// TwinCAT 3 PLC project DeviceLib
// Title: IBF_Device
// Company: Industrial Brains B.V.
// ProjectVersion: 0.0.0.0
// ProgramVersion: 3.1.4022.4
// CompilerDefines: InclSerialCom := 'true'
// libraries:
//   IBF_Utilities, * (Industrial Brains B.V.)
//   Tc2_Math, * (Beckhoff Automation GmbH)
//   Tc2_MC2, * (Beckhoff Automation GmbH)
//   Tc2_MC2_Drive, * (Beckhoff Automation GmbH)
//   Tc2_Standard, * (Beckhoff Automation GmbH)
// project tree:
//   Actuators/Cylinder/DataTypes/ E_CylinderCmd.TcTLEO, E_ValveResetState.TcTLEO
//   Actuators/Cylinder/DataTypes/ManualControls/ UDT_ManualValveControl.TcDUT
//   Actuators/Cylinder/Functions/ Fb_DevCylWithFbk.TcPOU, FB_DevValve.TcPOU
//   Axis/DataTypes/ E_AxisCmd.TcTLEO, UDT_AxisData.TcDUT, UDT_AxVal.TcDUT, UDT_ManualAxisCtrl.TcDUT
//   Axis/FunctionBlocks/Analog/ FB_DevAnalogAxis.TcPOU, ST_ManualAnalogAxisCtrl.TcDUT (not stored)
//   Axis/FunctionBlocks/ServoHybrid/ FB_DevBasicACAxis.TcPOU, FB_DevHybridAc.TcPOU
//   Axis/FunctionBlocks/Servo/ Fb_DevAxis.TcPOU
//   Axis/FunctionBlocks/TwoVelocityControl/DataTypes/ st_ManualDigitalMotorControl.TcDUT (not stored)
//   Axis/FunctionBlocks/TwoVelocityControl/ FB_DevTwoVelocityAxis.TcPOU
//   Axis/Interface/ iTwoDirectionalMotor.TcIO (not stored), iTwoDirectionalMotorWithFast.TcIO (not stored)
//   BaseFunctions/ FB_DevBase.TcPOU, UDT_DevManualCtrl.TcDUT
//   Buttons/Functions/ FB_DevHMIButton.TcPOU, FB_DevPushbuttonLight.TcPOU, FB_DevPushButton.TcPOU
//   CounterCards/FunctionBlocks/KL1512/ FB_DevKL1512.TcPOU
//   CounterCards/FunctionBlocks/KL5151/ FB_DevKL5151.TcPOU
//   CounterCards/Interfaces/ iCounter.TcIO
//   CounterCards/ st_ManualCounterControl.TcDUT
//   DevTypes/ E_Devices.TcTLEO
//   Encoders/FunctionBlocks/ FB_EncoderBase.TcPOU, FB_EncoderInput.TcPOU
//   GroupHandlers/ GVL_DevManual.TcGVL
//   GroupHandlers/ManualControlHandler/ FB_ManualController.TcPOU, UDT_DeviceID.TcDUT
//   HardwareDiagnostics/ FB_ELModuleDiag.TcPOU
//   Heaters/ FB_DevDoublePWM.TcPOU, FB_DevPWMGenerator.TcPOU
//   Lights/Functions/ Fb_DevLight.TcPOU
//   Outputs/AnalogOutputs/ FB_DevAnalogOutput.TcPOU, FB_DevAnalogOutputScaled.TcPOU
//   Outputs/DigitalOutputs/ FB_DevDigitalOutput.TcPOU
//   Sensors/AnalogInput/FunctionBlocks/ FB_DevAnalogInput.TcPOU, FB_DevAnalogInputScaled.TcPOU, FB_DevHDAnalogInAutoCalibrate.TcPOU, FB_DevAnalogInAutoCalibrate.TcPOU, FB_DevHDAnalogInputScaled.TcPOU, FB_DevHDAnalogInput.TcPOU
//   Sensors/DigitalSensor/FunctionBlocks/ Fb_DevDigitalInput.TcPOU, Fb_DevDigitalInputFunctions.TcPOU
//   Sensors/FootPedals/DataTypes/ E_FootpedalPos.TcTLEO
//   Sensors/FootPedals/FunctionBlocks/ FB_EfkaEB301A_FootPedal.TcPOU
//   Sensors/ModuleSpecific/EL3556_Loadcell/ Fb_DevEL3356_LoadCell.TcPOU (not stored)
//   Version/ Global_Version.TcGVL

// ---- Actuators/Cylinder/DataTypes/E_CylinderCmd.TcTLEO
(* cylinder commands *)
TYPE E_CylinderCmd :
(
	Cyl_Idle 		:= 0,// Jog Cylinder command Referance 0 Idle (wait for command)
	Cyl_Init 		:= 1,// Jog Cylinder command Referance 1 initialize Cylinder
	Cyl_Enable 		:= 2,// Jog Cylinder command Referance 2 enable
	Cyl_Disable 	:= 3,// Jog Cylinder command Referance 3 disable
	Cyl_Reset 		:= 4,// Jog Cylinder command Referance 4 reset
	Cyl_Hold 		:= 5,// Jog Cylinder command Referance 5 hold
	Cyl_Teach 		:= 6,// Jog Cylinder command Referance 6 teach timeout settings
	Cyl_Calculate 	:= 7,// Jog Cylinder command Referance 7 calculate timeout settings from parameters
	Cyl_Expand 		:= 8,// Jog Cylinder command Referance 8 expand
	Cyl_Retract 	:= 9 // Jog Cylinder command Referance 9 retract
);
END_TYPE

// ---- Actuators/Cylinder/DataTypes/ManualControls/UDT_ManualValveControl.TcDUT
TYPE UDT_ManualValveControl extends UDT_DevManualCtrl:
STRUCT
	// Device commands
	bCmdOpen	: BOOL	; // open valve 
	bCmdClose	: BOOL	; // Close valve
	bCmdTeach	: BOOL	; // Teach valve
END_STRUCT
END_TYPE

// ---- Axis/DataTypes/E_AxisCmd.TcTLEO
(* axis command structure *)
TYPE E_AxisCmd :
(
	Ax_Idle 		:= 0,// Axis command Referance 0 Axis Idle
	Ax_Init 		:= 1,// Axis command Referance 1 Initialize axis
	Ax_Enable 		:= 2,// Axis command Referance 2 Enable
	Ax_Disable 		:= 3,// Axis command Referance 3 Disable
	Ax_Reset 		:= 4,// Axis command Referance 4 Reset
	Ax_Hold 		:= 5,// Axis command Referance 5 Hold
	Ax_Home 		:= 6,// Axis command Referance 6 Home
	Ax_JogFwd 		:= 7,// Axis command Referance 7 Jog Forward
	Ax_JogRev 		:= 8,// Axis command Referance 8 Jog Reverse
	Ax_MoveRelative := 9,// Axis command Referance 9 Move axis relative
	Ax_MoveAbs 		:= 10,// Axis command Referance 11 Move absolute reverse
	Ax_MoveModulo 	:= 11,// Axis command Referance 11 Move Module
	Ax_MoveVeloFwd 	:= 12,// Axis command Referance 12 Move velocity forward
	Ax_MoveVeloRev 	:= 13,// Axis command Referance 13 Move velocity reverse
	Ax_HardStop 	:= 14,// Axis command Referance 14 hard stop or emergency stop
	Ax_SoftStop 	:= 15,// Axis command Referance 15 soft stop after motion command
	Ax_GearSlave 	:= 16,// Axis command Referance 16 gear axis as slave
	Ax_GearSlaveDyn	:= 17,// Axis command Referance 17 gear axis as slave dynamic
	Ax_GearOutSlave := 18,// Axis command Referance 18 gear out from Master axis 
	Ax_Maintenance	:= 50 // Axis Command referance 50 maintenance mode, axis enabled with no command active
);
END_TYPE

// ---- Axis/DataTypes/UDT_AxisData.TcDUT
TYPE UDT_AxisData:
STRUCT
	// ===== Axis name =====
		AxisName	: STRING 	; // Name of the axis (used for fault handling and identification)
		AxisNumber	: INT		; // Axis number 

	// ===== Fault data =====
		Message			: UDT_Fault 	; // Message data from Cylinder
		MessageActive	: BOOL			; // Message is active
		ErrorActive 	: BOOL 			;	// Axis in error state

	// ===== Axis Commands =====
		// ***** Enable command	*****
			CmdEnable		: BOOL 		; // Command enable axis
		// ***** Active commands *****
			AxisCmd			: E_AxisCmd ; // Axis command
			AxisSafeCmd		: E_AxisCmd	; // Axis safe command
			AxisAct			: E_AxisCmd ; // Axis Active status
		// ***** Command Modes *****
			CmdHomingMode 	: MC_HomingMode ; // Homing Mode ( MC_DefaultHoming, MC_Direct, MC_ForceCallibration, MC_ResetCallibration)
			CmdJogMode		: E_JogMode 	;
			CmdBuffermode	: MC_BufferMode	; // Buffermode used for command transition 	 
	// ===== Axis Safe commands =====
		SafeCmdLimitVelo: BOOL 	; // safe command limit velocity
		SafeCmdVelocity	: LREAL ; // Safe command velocity
		SafeCmdStop		: BOOL 	; // Stop command from safety or collision detection		
		SafeVeloLimit	: LREAL ; // safe velocity limit (link to FPAR)
	// ===== Status indication active =====
		ActHoming	: BOOL ; // Axis is homing
		ActBusy		: BOOL ; // Axis is Busy 
		ActMoving	: BOOL ; // Axis is moving
		ActAtVelo	: BOOL ; // Axis is at command velocity (only when written in Move velocity mode)

	// ===== Status indication done  =====
		FcoInit		: BOOL ; // Axis is initialised
		FcoIdle		: BOOL ; // Axis is idle enable required
		FcoEnabled	: BOOL ; // Axis is enabled
		FcoHomed	: BOOL ; // Axis is homed
		FcoGeared	: BOOL ; // Axis is geared to master axis
		FcoHeld		: BOOL ; // Axis is holding
		FcoStopped	: BOOL ; // Axis is stopped
		FcoReset	: BOOL ; // Axis reset done
		FcoReady 	: BOOL ; // Axis is ready for command
		FcoAtCmdPos	: BOOL ; // Axis is at command position (tol 0.2 deg)
		FcoCmdActive: BOOL ; // Axis new command values are active
		
	// ===== Move values =====
		Pos			: UDT_Axval	; // possition values (0 = infinite)
		Velocity 	: UDT_AxVal	; // Velocity values
		Accel		: UDT_Axval ; // Aceleration values
		Decel		: UDT_Axval ; // Deceleration values
		Torque		: UDT_Axval ; // Torque values
		EncTurnoverVal	: DINT 	; // Encoder turnover value
		TimeDisableDelay : TIME ; // Time off delay after axis move command (remove enable)
		
	// ===== Config Bits =====
		IcfCommandSpeedRpm	: BOOL ; // input speeds in Rpm
		IcfEnableForward 	: BOOL ; // Enable forward motion
 		IcfEnablereverse	: BOOL ; // Enable reverse motion
		IcfContinuous		: BOOL ; // continuous motion possible (no endpoint)
		IcfAlwaysEnable		: BOOL ; // 1 = Axis always enabled, 0 = Axis disabled at Idle 
		
	// ===== Master Axis =====
		MasterAxisRef	: REFERENCE TO AXIS_REF ; // Master axis reference (if applicable)
		GearMasterRev	: UINT	:= 1	; // Master Axis Gearing revolutions (Denominator)
		GearSlaveRev	: LREAL	:= 1	; // Slave Axis gearing revolutions (numerator)	
		ReverseSlave	: BOOL 	; // Reverse slave axis relative to master
		 
END_STRUCT
END_TYPE

// ---- Axis/DataTypes/UDT_AxVal.TcDUT
TYPE UDT_AxVal :
STRUCT
	// ***** Velocity settings *****
		HardMax		: LREAL 	; // Hardware maximum set absolute maximum
		ManMax 		: LREAL		; // Manual maximum percentage of hardware max
		AutoMax		: LREAL		; // Automatic maximum percentage of hardware max
		HomeMax		: LREAL 	; // Homing maximum percentage of hardware max
		CmdVal		: LREAL 	; // Commanded value
		SafeVal		: LREAL		; // Command value after safety check
		PrevVal		: LREAL		; // previous command value 
		ActVal		: LREAL		; // Actual value
		ActModulo	: LREAL		; // [deg] Modulo position
		RefVal		: LREAL 	; // referance value (basic setting or home) 
END_STRUCT
END_TYPE

// ---- Axis/DataTypes/UDT_ManualAxisCtrl.TcDUT
TYPE UDT_ManualAxisCtrl :
STRUCT
	bCmdJogForward	: 	BOOL 		; // command jog forward
	bCmdJogReverse	: 	BOOL 		; // command jog reverse
	bCmdInching		: 	BOOL 		; // Command move relative Distance
	bCmdToPos		: 	BOOL 		; // command move to absolute position (only moving when active)
	bCmdHome		: 	BOOL 		; // Command home axis
	fPosition		:	LREAL 		; // target position
	fDistance		:	LREAL 		; // target position
	fVelocity		: 	LREAL 		; // Maximum velocity [units/sec]
END_STRUCT
END_TYPE

// ---- BaseFunctions/UDT_DevManualCtrl.TcDUT
TYPE UDT_DevManualCtrl :
STRUCT
END_STRUCT
END_TYPE

// ---- CounterCards/st_ManualCounterControl.TcDUT
TYPE st_ManualCounterControl :
STRUCT
	bManSetValue 	: BOOL ; // Set value from manual control
	nManValue		: UDINT; // Manual value
END_STRUCT
END_TYPE

// ---- DevTypes/E_Devices.TcTLEO
{attribute 'qualified_only'}
{attribute 'strict'}
{attribute 'To String'}
TYPE E_Devices :
(
	Undefined,
	Valve,
	Cylinder,
	Axis,
	PushButtonLight,
	DigitalSensor,
	AnalogSensor,
	DigitalOut,
	AnalogOut,
	PWMController,
	DoublePWMController,
	Encoder,
	AnalogAxis,
	TwoVelocityAxis,
	KL5151
)INT;
END_TYPE

// ---- GroupHandlers/ManualControlHandler/UDT_DeviceID.TcDUT
TYPE UDT_DeviceID :
STRUCT
	sName			: STRING	; // device name
	sType			: STRING	; // Type of device [string for visu]
	pFunction		: POINTER TO FB_DevBase ; // Pointer to the device
END_STRUCT
END_TYPE

// ---- Actuators/Cylinder/DataTypes/E_ValveResetState.TcTLEO
{attribute 'qualified_only'}
{attribute 'strict'}
TYPE E_ValveResetState :
(
	Res_Idle 		:= 0,
	Res_Closed		:= 1,
	Res_Open		:= 2
);
END_TYPE

// ---- Sensors/FootPedals/DataTypes/E_FootpedalPos.TcTLEO
{attribute 'qualified_only'}
{attribute 'strict'}
TYPE E_FootpedalPos :
(
	eReverse2 	:= -2,
	eReverse1 	:= -1,
	eIdle		:= 0,
	eForward0	:= 1,
	eForward1	:= 2,
	eForward2	:= 3,
	eForward3	:= 4,
	eForward4	:= 5,
	eForward5	:= 6,
	eForward6	:= 7,
	eForward7	:= 8,
	eForward8	:= 9,
	eForward9	:= 10,
	eForward10	:= 11,
	eForward11	:= 12,
	eForward12	:= 13,
	eFalse			
) INT; 
END_TYPE
//  eReverse2 = '-2'
//  eReverse1 = '-1'

// ---- GroupHandlers/GVL_DevManual.TcGVL
{attribute 'qualified_only'}
VAR_GLOBAL
	fbManualControler	: FB_ManualController ; // Default Manual control function for devices (not called implicitly) 
	bManualModeActive	: BOOL ; // System manual mode is active
END_VAR
VAR_GLOBAL CONSTANT
	nMAXDEVCOUNT		: UDINT  := 100		; // Maximum number of devices 
END_VAR

// ---- Version/Global_Version.TcGVL
{attribute 'TcGenerated'}
{attribute 'no-analysis'}
{attribute 'linkalways'}
// This function has been automatically generated from the project information.
VAR_GLOBAL CONSTANT
	{attribute 'const_non_replaced'}
	stLibVersion_IBF_Device : ST_LibVersion := (iMajor := 0, iMinor := 0, iBuild := 0, iRevision := 0, nFlags := 0, sVersion := '0.0.0.0');
END_VAR

// ---- CounterCards/Interfaces/iCounter.TcIO
INTERFACE iCounter

METHOD PUBLIC CmdReset : BOOL
END_METHOD

METHOD PUBLIC CmdSetValue : BOOL
VAR_INPUT
	Value : UDINT ;
END_VAR
END_METHOD

PROPERTY PUBLIC CountValue : UDINT
GET
END_GET
END_PROPERTY

END_INTERFACE

// ---- GroupHandlers/ManualControlHandler/FB_ManualController.TcPOU
{attribute 'reflection'}
FUNCTION_BLOCK FB_ManualController
VAR_INPUT
	bReset 			: BOOL 		:= FALSE ; // (auto linked) reset selected device 
END_VAR
VAR_OUTPUT
	eDevType		: INT		:= E_Devices.Undefined	; // Selected device type
	bManual			: BOOL 		:= FALSE ; // selected device is in manual state
	bErroractive	: BOOL 		:= FALSE ; // Device error is active
	sDeviceState	: STRING	:= '' 	; // Dselected device fault message
END_VAR
VAR
	nNumberOfDevices	: UDINT := 0 	; // number of devices in manual array 
	
	bManualActive		: BOOL 	:= FALSE ; // Manual control mode is activated
	bDisableManualInputs: BOOL 	:= TRUE 	; // disable device manual inputs
	
	pDevValve			: POINTER TO FB_DevValve				; // Device pointer to valve
	pDevCylinder		: POINTER TO Fb_DevCylWithFbk 			; // Device pointer to cylinder with manual 
	pDevAxis			: POINTER TO Fb_DevAxis 				; // device pointer to Axis 
	pDevPBL				: POINTER TO FB_DevPushbuttonLight		; // Device pointer to puschbutton light
	pDevDigitalInput	: POINTER TO Fb_DevDigitalInputFunctions; // device pointer to digital input
	pDevAnalogInput		: POINTER TO FB_DevAnalogInput			; // Device pointer to analog input
	pDevAnalogOut		: POINTER TO FB_DevAnalogOutput			; // Device pointer to analog output
	pDevDigitalOut		: POINTER TO FB_DevDigitalOutput		; // Device pointer to digital output
	pDevPWMController	: POINTER TO FB_DevPWMGenerator			; // Device pointer to PWM controller
	pDevDoublePWM		: POINTER TO FB_DevDoublePWM			; // Device pointer to Double PWM controller
	pDevEncoder			: POINTER TO FB_EncoderBase				; // Device Pointer to encoder Base
	pDevAnalogAxis		: POINTER TO FB_DevAnalogAxis			; // Device pointer to analog axis control
	
	{attribute 'analysis' := '-33'}
	fbNodevice			: FB_DevBase ;
	stNoDevice			: UDT_DeviceID := (sName := 'No device', sType := TO_STRING(E_Devices.Undefined), pFunction := ADR(fbNodevice)); 
	arDeviceArray		: ARRAY [0..GVL_DevManual.nMAXDEVCOUNT] OF UDT_DeviceID := [stNoDevice]	; // Array of Devices for manual control
	nCmdLookupindex		: UDINT := 0; // Index number in array
	i					: UDINT := 0; // Index pointer to array
END_VAR

GVL_DevManual.bManualModeActive := bManualActive ;
IF bManualActive THEN 
	// insert a device 
	ExecSelectDevice();
END_IF

METHOD PUBLIC CmdAddDevice : BOOL
VAR_INPUT
	refToDevice	: REFERENCE TO FB_DevBase ;
END_VAR
VAR
	bDevAdded	: BOOL ;
END_VAR
// Check if device is not already in the array 
FOR i:= 0 TO nNumberOfDevices DO 
	IF arDeviceArray[i].sName = refToDevice.sName THEN 
		bDevAdded := TRUE ;
	END_IF 
END_FOR

// If device is not found add device to the list
IF NOT bDevAdded THEN 
	nNumberOfDevices := LIMIT(0, nNumberOfDevices + 1 ,GVL_DevManual.nMAXDEVCOUNT)	;
	arDeviceArray[nNumberOfDevices].sType 		:= TO_STRING(refToDevice.eDevType)	;
	arDeviceArray[nNumberOfDevices].sName		:= refToDevice.sName	;
	arDeviceArray[nNumberOfDevices].pFunction 	:= ADR(refToDevice)		;	
	bDevAdded := TRUE ;
END_IF

CmdAddDevice := bDevAdded ;
END_METHOD

METHOD PRIVATE ExecSelectDevice : BOOL
VAR_INPUT
END_VAR
// Select active manual device
bDisableManualInputs := NOT arDeviceArray[nCmdLookupindex].pFunction^.bManual ; 
IF bManualActive THEN 
	arDeviceArray[nCmdLookupindex].pFunction^.CmdManual(); 
END_IF

CASE arDeviceArray[nCmdLookupindex].pFunction^.eDevType OF
	E_Devices.Valve			:
		pDevValve 			:= arDeviceArray[nCmdLookupindex].pFunction ;
	E_Devices.Cylinder		:
		pDevCylinder		:= arDeviceArray[nCmdLookupindex].pFunction ;
	E_Devices.Axis 			:
		pDevAxis			:= arDeviceArray[nCmdLookupindex].pFunction ;
	E_Devices.PushButtonLight :
		pDevPBL				:= arDeviceArray[nCmdLookupindex].pFunction ;
	E_Devices.DigitalSensor :
		pDevDigitalInput	:= arDeviceArray[nCmdLookupindex].pFunction ;
	E_Devices.AnalogSensor 	:
		pDevAnalogInput 	:= arDeviceArray[nCmdLookupindex].pFunction ;
	E_Devices.DigitalOut	:
	 	pDevDigitalOut		:= arDeviceArray[nCmdLookupindex].pFunction ;
	E_Devices.AnalogOut		:
		pDevAnalogOut		:= arDeviceArray[nCmdLookupindex].pFunction ;
	E_Devices.PWMController	:
		pDevPWMController	:= arDeviceArray[nCmdLookupindex].pFunction ;
	E_Devices.DoublePWMController :
		pDevDoublePWM		:= arDeviceArray[nCmdLookupindex].pFunction ;
	E_Devices.Encoder :
		pDevEncoder			:= arDeviceArray[nCmdLookupindex].pFunction ;
	E_Devices.AnalogAxis:
		pDevAnalogAxis		:= arDeviceArray[nCmdLookupindex].pFunction ;
	ELSE
		;
END_CASE

// Set device command 
IF bReset THEN 
	bReset R= arDeviceArray[nCmdLookupindex].pFunction^.CmdReset();
END_IF

// Set device state feedback
bManual 		:= arDeviceArray[nCmdLookupindex].pFunction^.bManual ;
bErroractive	:= arDeviceArray[nCmdLookupindex].pFunction^.bErrorActive ;
sDeviceState	:= arDeviceArray[nCmdLookupindex].pFunction^.sActiveState ;

// Set device screen control 
eDevType := arDeviceArray[nCmdLookupindex].pFunction^.eDevType ;
END_METHOD

END_FUNCTION_BLOCK

// ---- Actuators/Cylinder/Functions/FB_DevValve.TcPOU
{attribute 'reflection'}
FUNCTION_BLOCK PUBLIC FB_DevValve EXTENDS FB_DevBase
VAR_INPUT
	// Manual control 
	stManualCtrl	: UDT_ManualValveControl ;
END_VAR
VAR_OUTPUT
	// ===== Status indicators =======
	bFco_Closed		:	BOOL := FALSE ;
	bFco_Open		: 	BOOL := FALSE ;
	fTimeToOpen		: 	LREAL ;
	fTimeToClose	: 	LREAL ;
END_VAR
VAR
	// Pararmeters
		stParTimeToClose	: Udt_Parameter := (fValue := 50) ; // time to close parameter
		stParTimeToOpen		: Udt_Parameter	:= (fValue := 50) ; // Time to open parameter
	// Hardware links 
		q_Open			AT %Q* : BOOL := FALSE 	; // Open valve
		q_Close 		AT %Q* : BOOL := FALSE	; // Close valve
	// Internal commands
		bCmdClose 	: BOOL := FALSE ; // close valve 
		bCmdOpen	: BOOL := FALSE ; // Open valve
		bCmdHold	: BOOL := FALSE ; // Hold valve status change
	// Time functions 
		fbTOnClose	: TON	; // Timer for valve close
		FbTOnOpen	: TON 	; // Timer for valve Open
		fbTimerSwitchDir: TON ; // Time for teach function switch direction 
	// reset and safe state
		eResetState		: E_ValveResetState := 0		; // Cylinder reset state variable (default is idle) 
		eSafeState		: E_ValveResetState	:= 0		; // Valve safe state
END_VAR

// set device type
IF eDevType = E_Devices.Undefined THEN 
	eDevType := E_Devices.Valve ;
END_IF

// Call base function
	SUPER^(refFbFault := refFbFault);

// ===== hold all actions if not initialized ======
IF NOT bInitOk THEN
	RETURN;
END_IF 

// ====== Set Outputs =======
	ExecSetOutPuts();

// ===== collect feedback ======
	ExecSetFeedback();

METHOD PUBLIC CmdClose : BOOL // close valve or retract cylinder
VAR_INPUT
END_VAR
IF bCmdManual THEN 
	RETURN;
END_IF

// ====== Set close command if enabled ======
	bCmdClose 	:= TRUE	;		
	bCmdOpen 	:= FALSE;

// ====== Check if command is blocked =====
	bBlockedCommand := bCmdHold;
	
// ===== Set feedback ======
	CmdClose := bFco_Closed ;
END_METHOD

METHOD PUBLIC CmdHold : BOOL
VAR_INPUT
END_VAR
// ====== set hold command =====
	bCmdHold := TRUE ;

CmdHold := bBlockedCommand ;
END_METHOD

METHOD PUBLIC CmdManual : BOOL
VAR_IN_OUT
END_VAR
// Enable manual commands
bCmdManual S= TRUE ;

// execute manual command 
	IF stManualCtrl.bCmdOpen THEN 
		bCmdClose 	:= FALSE;		
		bCmdOpen 	:= TRUE	;
	ELSIF stManualCtrl.bCmdClose THEN 
		bCmdClose 	:= TRUE	;		
		bCmdOpen 	:= FALSE;
	ELSIF stManualCtrl.bCmdTeach THEN
		CmdTeach ();
	END_IF
END_METHOD

METHOD PUBLIC CmdOpen : BOOL // Open valve or retract cylinder
VAR_INPUT
END_VAR
IF bCmdManual THEN 
	RETURN;
END_IF

// ====== Set open command if enabled ======
	bCmdClose 	:= FALSE;		
	bCmdOpen 	:= TRUE	;

// ====== Check if command is blocked =====
	bBlockedCommand := bCmdHold;
	
// ===== Set feedback ======
	CmdOpen := bFco_Open ;
END_METHOD

METHOD PUBLIC CmdReset : BOOL
VAR_INPUT
END_VAR
// ====== Set outputs according to reset state =======
	IF bEnable THEN 
		CASE eResetState OF 
			E_ValveResetState.Res_Idle:
				bCmdClose 	:= FALSE;		
				bCmdOpen 	:= FALSE;
			E_ValveResetState.Res_Closed:
				bCmdClose 	:= TRUE	;		
				bCmdOpen 	:= FALSE;
			E_ValveResetState.Res_Open:
				bCmdClose 	:= FALSE;		
				bCmdOpen 	:= TRUE	;
		ELSE
			;
		END_CASE
	END_IF
// ======= Reset Error bit ======
	bErrorActive 	:= FALSE;
	bBussy			:= FALSE;
	
// ======= set feedback =======
	CmdReset := TRUE ;
END_METHOD

METHOD PUBLIC CmdSafeStop : BOOL
VAR_INPUT
END_VAR
bCmdOpen := FALSE ;
bCmdClose:= FALSE ;

CASE eSafeState OF 
	E_ValveResetState.Res_Idle:
		q_Close := FALSE ;
		q_Open  := FALSE ;
		bIsSafe := TRUE ;
	E_ValveResetState.Res_Closed:
		q_Close := TRUE ;
		q_Open  := FALSE ;
		bIsSafe := bFco_Closed OR NOT bFco_Open ;
	E_ValveResetState.Res_Open:
		q_Close := FALSE ;
		q_Open  := TRUE ;
		bIsSafe := bFco_Open OR NOT bFco_Closed;
END_CASE

CmdSafeStop := bIsSafe OR NOT bInitOk ;
END_METHOD

METHOD PUBLIC CmdTeach : BOOL
VAR_INPUT
END_VAR
// ====== teach cylinder from hardware inputs ======
	fbTimerSwitchDir(PT:= T#1S); 
// ===== Start test loop =====
IF bFco_Closed AND fbTimerSwitchDir.Q THEN
	bCmdClose 			:= FALSE;
	bCmdOpen 			:= TRUE ;
	fbTimerSwitchDir.IN	:= FALSE; 
ELSIF bFco_Open AND fbTimerSwitchDir.Q THEN
	bCmdClose 			:= TRUE ;
	bCmdOpen 			:= FALSE;
	fbTimerSwitchDir.IN	:= FALSE; 
ELSIF NOT bCmdClose AND NOT bCmdOpen THEN 
	bCmdClose 			:= TRUE ;
	bCmdOpen 			:= FALSE;
END_IF

// ====== start timing ========
	IF bCmdClose AND bFco_Closed THEN 
		fbTimerSwitchDir.IN := TRUE 		;
	ELSIF bCmdOpen AND bFco_Open THEN 
		fbTimerSwitchDir.IN := TRUE 		;
	END_IF
END_METHOD

METHOD PROTECTED ExecSetFeedback : BOOL
VAR_INPUT
END_VAR
// ====== Set timers =======
	fbTOnClose	(PT 	:= LREAL_TO_TIME(stParTimeToClose.fValue))	;
	FbTOnOpen	(PT		:= LREAL_TO_TIME(stParTimeToOpen.fValue))	;

// ====== Set timed feedback ======
	IF q_Close THEN 
		fbTOnClose.IN 	:= TRUE ;
		fbTOnopen.IN 	:= FALSE;
	ELSIF q_Open THEN 
		fbTOnClose.IN 	:= FALSE;
		FbTOnOpen.IN	:= TRUE ;
	ELSE 
		fbTOnClose.IN 	:= FALSE;
		FbTOnOpen.IN	:= FALSE;
	END_IF
	
// ====== set outputs =======
	bFco_Closed := fbTOnClose.Q ;
	bFco_Open	:= FbTOnOpen.Q	;
	bReady		:= bFco_Closed OR bFco_Open ;
	
// ====== Timer values =====
	fTimeToClose	:= stParTimeToClose.fValue;
	fTimeToOpen		:= stParTimeToOpen.fValue;
END_METHOD

METHOD PROTECTED ExecSetOutPuts : BOOL
VAR_INPUT
END_VAR
// ======= Set Outputs according to commands and check safety features =======
IF bSafetyOk THEN
	IF NOT bCmdHold AND (bEnable OR bCmdManual) THEN  
		q_Close	:= bCmdClose;
		q_Open	:= bCmdOpen	;
	END_IF
ELSE
	CASE eSafeState OF 
		E_ValveResetState.Res_Idle:
			q_Close	:= bFco_Closed;		
			q_Open 	:= bFco_Open;
		E_ValveResetState.Res_Closed:
			q_Close	:= TRUE	;		
			q_Open 	:= FALSE;
		E_ValveResetState.Res_Open:
			q_Close	:= FALSE;		
			q_Open 	:= TRUE	;
	END_CASE
	bCmdClose 	:= bFco_Closed 	;
	bCmdOpen	:= bFco_Open	;
	
END_IF

// Reset manual and hold commands
bCmdHold 	:= FALSE ;
bCmdManual 	:= FALSE ;
END_METHOD

METHOD PUBLIC Init : BOOL
VAR_INPUT
	// Messagedata 
	nId			: UDINT ; // Identification number of object
	nParentId	: UDINT ; // Id of higher level If aplicable (0 = no parent)

	// Command state
	eResetState		: E_ValveResetState := 0		; // Cylinder reset state variable (default is idle) 
	eSafeState		: E_ValveResetState	:= 0		; // Valve safe state
END_VAR
// ====== Set init to true =====
	bInitOk	:= TRUE ; 

// ====== Calculate device id =====
	bInitOk :=	ExecIdentifyDevice(nId,nParentId, E_ComponentTypes.Cylinder) AND bInitOk;
	
// ====== Set message information =======
	stFault.ComponentType	:= E_ComponentTypes.Cylinder 		;
	
// ====== Set outputs according to reset state =======
	THIS^.eResetState 	:= eResetState 	;
	THIS^.eSafeState	:= eSafeState	;	

	IF bEnable THEN 
		CASE eResetState OF 
			E_ValveResetState.Res_Idle:
				bCmdClose 	:= bFco_Closed	;		
				bCmdOpen 	:= bFco_Open	;
			E_ValveResetState.Res_Closed:
				bCmdClose 	:= TRUE;		
				bCmdOpen 	:= FALSE;
			E_ValveResetState.Res_Open:
				bCmdClose 	:= FALSE;		
				bCmdOpen 	:= TRUE ;
		END_CASE
	END_IF
// ======= Reset Error bit ======
	bErrorActive 	:= FALSE;
	bBussy			:= FALSE;

// ===== Set device type for manual control =====
	eDevType := E_Devices.Valve ;
	
// ===== configure parameters =====
	stParTimeToClose.fMinimum 		:= 0 		;
	stParTimeToClose.fMaximum		:= 60000 	;
	stParTimeToClose.nNumber 		:= nLocationId + 1;
	stParTimeToClose.sDiscription  	:= CONCAT( STR1 := sName, STR2 := 'avarage time it takes for the valve to close in miliseconds');
	stParTimeToClose.sName			:= CONCAT( STR1 := sName, STR2 := 'time to close');
	stParTimeToClose.sType			:= 'CPar';
	stParTimeToClose.sUnit			:= 'ms';

	stParTimeToOpen.fMinimum 		:= 0 		;
	stParTimeToOpen.fMaximum		:= 60000 	;
	stParTimeToOpen.nNumber 		:= nLocationId + 2;
	stParTimeToOpen.sDiscription  	:= CONCAT( STR1 := sName, STR2 := 'avarage time it takes for the valve to open in miliseconds');
	stParTimeToOpen.sName			:= CONCAT( STR1 := sName, STR2 := 'time to open');
	stParTimeToOpen.sType			:= 'CPar';
	stParTimeToOpen.sUnit			:= 'ms';
	
	// add parameters to handler 
	refFbParHandler.CmdAddParameter( refParameter := stParTimeToClose );
	refFbParHandler.CmdAddParameter( refParameter := stParTimeToOpen );

// Set feedback
Init := bInitOk;
END_METHOD

END_FUNCTION_BLOCK

// ---- BaseFunctions/FB_DevBase.TcPOU
{attribute 'reflection'}
FUNCTION_BLOCK PUBLIC FB_DevBase EXTENDS FB_FunctionBase
VAR_INPUT
	bEmbeded		: BOOL 	:= FALSE ; // Device is embedded into another device (not added to manual screen)
	// function references 
	refFbManualCtrl	: REFERENCE TO FB_ManualController := GVL_DevManual.fbManualControler	; // reference to manual handler
END_VAR
VAR_OUTPUT
	eDevType		: E_Devices		:= E_Devices.Undefined	; // Type of Device 	
END_VAR
VAR
	// Manual control variables
	bAddedToManual	: BOOL 	:= FALSE 	; // device is added tot manual control function 	
END_VAR

SUPER^(refFbFault := refFbFault);

// Add device to manual screen
IF NOT bEmbeded THEN 
	IF NOT bAddedToManual 
	AND sName <> '' 
	AND __ISVALIDREF(refFbManualCtrl)
	THEN 
		bAddedToManual S= refFbManualCtrl.CmdAddDevice(THIS^);
	END_IF
END_IF

METHOD PUBLIC CmdManual : BOOL
VAR_INPUT
END_VAR
bCmdManual := true ;
END_METHOD

METHOD PUBLIC CmdSafeStop : BOOL
VAR_INPUT
END_VAR
// check if device is safe
bIsSafe 	:= NOT bSafetyOk ;
CmdSafeStop := bIsSafe ;
END_METHOD

END_FUNCTION_BLOCK

// ---- Actuators/Cylinder/Functions/Fb_DevCylWithFbk.TcPOU
{attribute 'reflection'}
FUNCTION_BLOCK PUBLIC Fb_DevCylWithFbk EXTENDS FB_DevValve
VAR_INPUT
	bIcfFbkOpenPresent 	: BOOL := FALSE ; // Feedback for cylinder open is present 
	bIcfFbkClosedPresent: BOOL := FALSE ; // Feedback for Cylinder closed is present
	bIcfTimeChecked		: BOOL := TRUE 	; // Cylinder timing is checked = default true
	nMargin				: LREAL:= 10	; // % of tollerance in move speed 
END_VAR
VAR_OUTPUT
	// ===== Teach function =======
	bCmdCopyTimeParam 	: BOOL	:= FALSE 	;// Cylinder, Command to higher level copy toucht time to parameters
	bFeClosed			: BOOL 	:= FALSE	; // closed sensor falling edge
	bReClosed			: BOOL 	:= FALSE	; // closed sensor rising edge
	bFeOpen				: BOOL 	:= FALSE 	; // Open sensor falling edge
	bReOpen				: BOOL 	:= FALSE 	; // open sensor rising edge 
	bReOpenSlow         : BOOL  := FALSE    ; // rising edge, opening went too slow
	bReOpenFast         : BOOL  := FALSE    ; // rising edge, opening went too fast
	bReCloseSlow        : BOOL  := FALSE    ; // rising edge, closing went too slow
	bReCloseFast        : BOOL  := FALSE    ; // rising edge, closing went too fast
END_VAR
VAR	
	bFcoCalcDone	: BOOL := FALSE ; // Calculate timers done 
	
	stTimesClose	: Udt_TimerBandwith ; // Timer bandwith for cylinder close
	stTimesOpen		: Udt_TimerBandwith	; // Timer bandwitch for cylinder open 
	
	fbSensorClosed	: Fb_DevDigitalInputFunctions ; // Digital sensor function closed detection
	fbSensorOpen	: Fb_DevDigitalInputFunctions ; // Digital sensor function open detection
	
	fbTimerOpen		: TON ; // Timer for cylinder to open
	fbTimerClose 	: TON ; // Timer for cylinder to close
	fbTimerTeach	: TON ; // timer for teachin cylinder 

	rtCmdWriteParam	: R_TRIG ; // Write parameter rising edge trigger 
	// Simulation
	fbTimerSimOpen 	: TON 	; 
	fbTimerSimClose	: TON 	; 
	
	// Time Cylinder valid 
	bTriggerTimeClose	: BOOL ;
	bTriggerTimeOpen	: BOOL ;
END_VAR

// set device type
	IF eDevType = E_Devices.Undefined THEN 
		eDevType := E_Devices.Cylinder ;
	END_IF

// call base function 
	SUPER^(refFbFault := refFbFault);

// check for device init
	IF NOT bInitOk THEN
		RETURN;
	END_IF 

// ====== Check direction of movement =======
	ExecDirection();
	
// ====== Reset movement indicators =======
	bReOpenSlow  := FALSE;
	bReOpenFast  := FALSE;
	bReCloseSlow := FALSE;
	bReCloseFast := FALSE;

// ====== Check movement speed =======
	ExecTimeout();
	
// ====== Calculate timers =======
	CalcTimers();

METHOD PRIVATE CalcTimers : BOOL
VAR
END_VAR
IF stParTimeToClose.fValue = stTimesClose.Nominal AND stParTimeToOpen.fValue = stTimesOpen.Nominal AND bFcoCalcDone THEN 
	RETURN ;
ELSE
	bFcoCalcDone := FALSE ;
END_IF
 
// ====== Calculate close times ======
	stTimesClose.Nominal 	:= stParTimeToClose.fValue ;
	stTimesClose.Maximum 	:= stParTimeToClose.fValue * (1 + (nMargin / 100));
	stTimesClose.Minimal 	:= stParTimeToClose.fValue * (1 - (nMargin / 100));

// ====== Calculate open times ======
	stTimesOpen.Nominal 	:= stParTimeToOpen.fValue ;
	stTimesOpen.Maximum 	:= stParTimeToOpen.fValue * (1 + (nMargin / 100));
	stTimesOpen.Minimal 	:= stParTimeToOpen.fValue * (1 - (nMargin / 100));
	
// ====== Set feedback =======
	bFcoCalcDone := TRUE ;

// ===== send write parameters command ======	
	rtCmdWriteParam(CLK := bFcoCalcDone);
	bCmdCopyTimeParam := rtCmdWriteParam.Q	;
END_METHOD

METHOD PUBLIC CmdSimulate : BOOL
VAR_INPUT
	bFbkReverse		: BOOL := FALSE ; 
	tTimeSimOpen	: TIME := T#1S 	;
	tTimeSimClose	: TIME := T#1S 	;  
END_VAR
// Run timers when cylinder is active 
	fbTimerSimOpen	(IN := q_Open	, PT := tTimeSimOpen);
	fbTimerSimClose	(IN := q_Close	, PT := tTimeSimClose);

// set feedback sensors to simulate
	fbSensorOpen.bCmdSimulate 	:= TRUE ;
	fbSensorClosed.bCmdSimulate := TRUE ;

// set simulated feedback state 
	IF bFbkReverse THEN 
		fbSensorClosed.bSimState:= fbTimerSimOpen.Q 	;
		fbSensorOpen.bSimState	:= fbTimerSimClose.Q 	; 	
	ELSE 
		fbSensorClosed.bSimState:= fbTimerSimClose.Q 	;
		fbSensorOpen.bSimState	:= fbTimerSimOpen.Q 	; 	
	END_IF
END_METHOD

METHOD PUBLIC CmdTeach : BOOL
VAR_INPUT
END_VAR
// ====== turn off time check function until new calculation cycle =======
	bFcoCalcDone := false ;

// ====== teach cylinder from hardware inputs ======
	fbTimerTeach	(PT:= T#60S);
	fbTimerSwitchDir(PT:= T#1S); 
// ====== time cylinder cycles ======
	// ===== Start test loop =====
	IF bFco_Closed AND fbTimerSwitchDir.Q THEN
		bCmdClose 			:= FALSE;
		bCmdOpen 			:= TRUE ;
		fbTimerSwitchDir.IN	:= FALSE; 
		fbTimerTeach.IN 	:= TRUE ;
	ELSIF bFco_Open AND fbTimerSwitchDir.Q THEN
		bCmdClose 			:= TRUE ;
		bCmdOpen 			:= FALSE;
		fbTimerSwitchDir.IN	:= FALSE; 
		fbTimerTeach.IN 	:= TRUE ;
	ELSIF NOT bCmdClose AND NOT bCmdOpen THEN 
		bCmdClose 			:= TRUE ;
		bCmdOpen 			:= FALSE;
		fbTimerTeach.IN 	:= TRUE ;
	END_IF

// ====== start timing ========
	IF bCmdClose AND bFco_Closed THEN 
		IF fbTimerTeach.IN THEN
			stParTimeToClose.fValue 	:= TIME_TO_LREAL(fbTimerTeach.ET);
		END_IF
		fbTimerSwitchDir.IN := TRUE 		;
		fbTimerTeach.IN 	:= FALSE 		;
	ELSIF bCmdOpen AND bFco_Open THEN 
		IF fbTimerTeach.IN THEN
			stParTimeToOpen.fValue		:= TIME_TO_LREAL(fbTimerTeach.ET);
		END_IF
		fbTimerSwitchDir.IN := TRUE 		;
		fbTimerTeach.IN 	:= FALSE 		;
	END_IF
END_METHOD

METHOD PRIVATE ExecDirection : BOOL
VAR_INPUT
END_VAR
// ===== Check direction commands =====
 	IF q_Close AND fbSensorOpen.bReStatus AND NOT q_Open THEN
		stFault.Active			:= TRUE ;
		stFault.MessageNumber	:= E_MessageNumbers.CF_WrongDirection 	;
		stFault.Discription		:= CONCAT( sName,' Cylinder Opening instead of closing');
		stFault.FaultType		:= E_FaultTypes.CF 					;
		bErrorActive			:= TRUE 								;
	ELSIF q_Open AND fbSensorClosed.bReStatus AND NOT q_close THEN
		stFault.Active			:= TRUE ;
		stFault.MessageNumber	:= E_MessageNumbers.CF_WrongDirection 	;
		stFault.Discription		:= CONCAT( sName,' Cylinder closing instead of opening');
		stFault.FaultType		:= E_FaultTypes.CF 					;
		bErrorActive			:= TRUE 								;
	END_IF
END_METHOD

METHOD PROTECTED ExecSetFeedback : BOOL
VAR_INPUT
END_VAR
{warning disable C0371}
// ====== Call sensor Open function =======
	IF bIcfFbkClosedPresent THEN 
		fbSensorClosed(refFbFault := refFbFault);
		bFco_Closed := fbSensorClosed.bFcoInputActive ;
		bFeClosed 	:= fbSensorClosed.bFeStatus ;
		bReClosed 	:= fbSensorClosed.bReStatus ;
	ELSE 
		fbTOnClose	(IN 	:= q_Close, PT 	:= LREAL_TO_TIME(stParTimeToClose.fValue))	;
		bFco_Closed := fbTOnClose.Q ;
	END_IF

// ====== Call sensor Close function =======
	IF bIcfFbkOpenPresent THEN 
		fbSensorOpen(refFbFault := refFbFault) 	;
		bFco_open 	:= fbSensorOpen.bFcoInputActive ;
		bFeOpen		:= fbSensorOpen.bFeStatus;
		bReOpen		:= fbSensorOpen.bReStatus;
	ELSE 
		FbTOnOpen	(IN 	:= q_Open, PT 	:= LREAL_TO_TIME(stParTimeToOpen.fValue))	;
		bFco_Open := FbTOnOpen.Q ;
	END_IF

{warning restore C0371}
// ====== set outputs =======
	bReady		:= bFco_Closed OR bFco_Open ;
END_METHOD

METHOD PRIVATE ExecTimeout : BOOL
VAR_INPUT
END_VAR
VAR
	nTimePassedMs : LREAL ;
END_VAR
IF bFcoCalcDone AND bIcfTimeChecked AND bEnable THEN 
// ====== Set triggers ======
	IF q_Close  AND bFco_Open THEN 
		bTriggerTimeClose := TRUE ;
	ELSIF q_Open OR bFco_Closed  THEN 
		bTriggerTimeClose := FALSE ;
	END_IF

	IF q_Open  AND bFco_Closed THEN 
		bTriggerTimeOpen := TRUE ;
	ELSIF q_Close OR bFco_Open THEN
		bTriggerTimeOpen := FALSE ;
	END_IF
ELSE
	bTriggerTimeClose 	:= FALSE ;
	bTriggerTimeOpen	:= FALSE ;
END_IF


//======= run timers =======
	IF bIcfFbkClosedPresent THEN 
		fbTimerClose(IN := q_Close AND bEnable, PT := LREAL_TO_TIME(stTimesClose.Maximum + 10));
	END_IF	
	
	IF bIcfFbkOpenPresent THEN 
		fbTimerOpen	(IN := q_Open AND bEnable , PT := LREAL_TO_TIME(stTimesOpen.Maximum + 10));
	END_IF

//====== Run timeout checks for cylinder close =======
	nTimePassedMs:= TIME_TO_LREAL(fbTimerClose.ET);
	
	IF bIcfFbkClosedPresent THEN 
		IF bTriggerTimeClose THEN 
			IF fbSensorClosed.bReStatus THEN 
				IF nTimePassedMs < stTimesClose.Minimal THEN 
					// send message to HMI 
					stFault.Active			:= TRUE 							;
					stFault.MessageNumber	:= E_MessageNumbers.CF_MoveToFast 	;
					stFault.Discription		:= CONCAT( sName, ' Cylinder closing to fast' )	;
					stFault.FaultType		:= E_FaultTypes.CF 					;
					bErrorActive			:= TRUE 							;
					bReCloseFast			:= TRUE                             ;
				END_IF
			ELSIF	nTimePassedMs > stTimesClose.Maximum  THEN
				// send message to HMI 
				stFault.Active			:= TRUE ;
				stFault.MessageNumber	:= E_MessageNumbers.CF_MoveToSlow		;
				stFault.Discription		:= CONCAT( sName,' Cylinder closing to Slow')	;
				stFault.FaultType		:= E_FaultTypes.CF 						;
				bErrorActive			:= TRUE 								;
				bReCloseSlow			:= TRUE                             	;
			END_IF
		END_IF
	END_IF	

//====== Run timeout checks for cylinder Open =======
	nTimePassedMs:= TIME_TO_REAL(fbTimerOpen.ET);

	IF bIcfFbkOpenPresent THEN 
		IF bTriggerTimeOpen THEN 
			IF fbSensorOpen.bReStatus THEN 
				IF nTimePassedMs < stTimesOpen.Minimal THEN 
					// send message to HMI 
					stFault.Active			:= TRUE ;
					stFault.MessageNumber	:= E_MessageNumbers.CF_MoveToFast 	;
					stFault.Discription		:= CONCAT( sName,' Cylinder Opening to fast')		;
					stFault.FaultType		:= E_FaultTypes.CF 					;
					bErrorActive			:= TRUE 							;
					bReOpenFast 			:= TRUE 							;
				END_IF
			ELSIF	nTimePassedMs > stTimesOpen.Maximum  THEN
				// send message to HMI 
				stFault.Active			:= TRUE ;
				stFault.MessageNumber	:= E_MessageNumbers.CF_MoveToSlow 	;
				stFault.Discription		:= CONCAT( sName,' Cylinder Opening to Slow')		;
				stFault.FaultType		:= E_FaultTypes.CF 					;
				bErrorActive			:= TRUE 							;
				bReOpenSlow 			:= TRUE 							;
			END_IF
		END_IF
	END_IF
END_METHOD

METHOD PUBLIC Init : BOOL
VAR_INPUT
	// Message location data
	nId			: UDINT ; // Identification number of object
	nParentId	: UDINT ; // Id of higher level If aplicable (0 = no parent)
	// Command state
	eResetState		: E_ValveResetState := 0		; // Cylinder reset state variable (default is idle) 
	eSafeState		: E_ValveResetState	:= 0		; // Valve safe state
END_VAR
bFcoCalcDone := FALSE;

// Enable sensor feedback
fbSensorClosed.bEmbeded := TRUE ;
fbSensorClosed.bEnable	:= TRUE ;
fbSensorClosed.Init	(	nId 		:= 0,
						nParentId 	:= nLocationId) ;

fbSensorOpen.bEmbeded := TRUE ;
fbSensorOpen.bEnable	:= TRUE ;
fbSensorOpen.Init	(	nId 		:= 1,
						nParentId 	:= nLocationId) ;

// Call feedback sensors 
ExecSetFeedback(); 

SUPER^.Init(nId, nParentId, eResetState, eSafeState);

// ===== Set device type for manual control =====
eDevType := E_Devices.Cylinder ;

bInitOk := fbSensorClosed.bInitOk 	AND bInitOk ;
bInitOk := fbSensorOpen.bInitOk		AND bInitOk ;
Init 	:= bInitOk ;
END_METHOD

END_FUNCTION_BLOCK

// ---- Sensors/DigitalSensor/FunctionBlocks/Fb_DevDigitalInputFunctions.TcPOU
{attribute 'reflection'}
FUNCTION_BLOCK PUBLIC Fb_DevDigitalInputFunctions EXTENDS Fb_DevDigitalInput
VAR_OUTPUT
	bFcoDelay			: BOOL			;// Digital sensor, Delayed input status (3 seconds) 
	bFeStatus			: BOOL			;// Digital sensor, Falling edge of input signal	
	bReStatus			: BOOL			;// Digital sensor, Rising edge of input signal
	bFcoFlipFlop		: BOOL			;// Digital sensor, feedback flip flop
	TetInputActive		: TIME			;// Digital sensor, Time elapsed while button is active
END_VAR
VAR
	// ***** Fucntion blocks *****
		FB_delIStatus	: TON	; // Timer function for delayed input status 
		FB_feIStatus	: F_TRIG; // generate falling edge pulse edge from Istatus
		FB_reIStatus	: R_TRIG; // generate falling edge pulse edge from Istatus
		FB_rsIStatus	: RS	; // Set Reset function for flip flop input
END_VAR

SUPER^(refFbFault := refFbFault);


// ====== process functions if enabled ======
	// ***** Set Delayed inputs and time elapsed ****
		FB_delIStatus(	IN:= bFcoInputActive,
						PT:= tDelay , 
						Q=> bFcoDelay , 
						ET=> TetInputActive 
					  ); // Generate delayed input status from push button input status
	// ***** Edge triggers *****
		FB_feIStatus(CLK:= bFcoInputActive , Q=> bFeStatus ); // generate falling edge pulse on pushbutton input
		FB_reIStatus (Clk := bFcoInputActive , Q => bReStatus); // Generate rising edge from push button input signal
	// ***** Flip Flop *****
		FB_rsIStatus(	SET:= bFeStatus AND NOT bFcoFlipFlop , 
						RESET1:= bFeStatus AND bFcoFlipFlop , 
						Q1=> bFcoFlipFlop 
					 ); // Generate set reset function from pushbutton input status

END_FUNCTION_BLOCK

// ---- Sensors/DigitalSensor/FunctionBlocks/Fb_DevDigitalInput.TcPOU
{attribute 'reflection'}
FUNCTION_BLOCK PUBLIC Fb_DevDigitalInput EXTENDS FB_DevBase 
VAR_INPUT
	tDelay				: TIME 	:= T#1S	;// Time before delayed signal becomes active 
	bCmdSimulate		: BOOL 	:= FALSE ;// Simulate sensor Input 
	bSimState			: BOOL 	:= FALSE ;// Simulated sensor state
	bIcfNormalyClosed	: BOOL  := FALSE ;// Hardware input is a normally closed contact
	ibSoftInput			: BOOL 			;// Software input (bFcoInputActive := 
END_VAR
VAR_OUTPUT
	bFcoInputActive		: BOOL 			;// Digital sensor, Button active state
END_VAR
VAR
	Istatus		AT 	%I* : BOOL			;// Digital sensor, Direct input status
END_VAR

// Set device type
IF eDevType = E_Devices.Undefined THEN 
	eDevType := E_Devices.DigitalSensor ;
END_IF

// Call base function
SUPER^(refFbFault := refFbFault);

// ***** Direct input when enabled *****
IF bEnable OR bCmdManual THEN 
	IF bCmdSimulate  THEN 
		bFcoInputActive := bSimState ;
		bCmdSimulate	:= FALSE ;  
	ELSIF bIcfNormalyClosed THEN
		bFcoInputActive := NOT Istatus OR ibSoftInput;
	ELSE
		bFcoInputActive := Istatus OR ibSoftInput ;
	END_IF
ELSE 
	bFcoInputActive := FALSE ;
END_IF

METHOD PUBLIC Init : BOOL
VAR_INPUT
	// Location data for messages  
	nId			: UDINT ; // Identification number of object
	nParentId	: UDINT ; // Id of higher level If aplicable (0 = no parent)
END_VAR
// ====== Set init to true =====
	bInitOk	:= TRUE ; 

// ====== Calculate device id =====
	bInitOk :=	ExecIdentifyDevice(nId,nParentId, E_ComponentTypes.DiInput) AND bInitOk;

	Init	:= true ;
END_METHOD

END_FUNCTION_BLOCK

// ---- Axis/FunctionBlocks/Servo/Fb_DevAxis.TcPOU
{attribute 'reflection'}
FUNCTION_BLOCK PUBLIC Fb_DevAxis EXTENDS FB_DevBase
VAR_INPUT
	// ===== General Function input =====
		fCmdAcc			: LREAL := 15000;
		fCmdDecc		: LREAL := 15000; 
	// ===== Master Axis =====
		refMasterAxis	: REFERENCE TO AXIS_REF ; // Master axis reference (if applicable)
		bReverseSlave	: BOOL 	:= FALSE; // Reverse slave axis relative to master
		fCmdGearRatio	: LREAL := 1 ; // Gear ratio Master/Slave (1/Ratio) 
	// Manual control reference
		stManualCtrl	: UDT_ManualAxisCtrl ;
END_VAR
VAR_OUTPUT
	// ====== State indications =======
		bHomed			: BOOL 	:= FALSE; 
		bError 			: BOOL 	:= FALSE;
		bStopped		: BOOL 	:= FALSE;
		bResetDone		: BOOL 	:= FALSE;
		bGearedAsSlave	: BOOL 	:= FALSE;
		bVelocityLimited: BOOL 	:= FALSE;  
		bIdle			: BOOL 	:= FALSE;
		fVelocity		: LREAL	:= 0	; // Axis velocity [rpm or units/sec] depending on config
		fActPosition	: LREAL := 0	; // Axis actual position [Units] depending on config	
		bReInTargetPos	: BOOL 	:= false; // rising edge axis is in position
	// ====== axis reference ======
		AxisRef			: AXIS_REF	; // Axis reference to hardware 
	// ====== Axis Settings ======
		fMaxVelo		: LREAL := 0 ; // Axis Maximum velocity
		fMaxAcc			: LREAL := 0 ; // Axis Maximum cceleration
		fMaxDec			: LREAL := 0 ; // axis Maxium deceleration 
	
//		fSafeVeloLimit	: LREAL	:= 200; // Safe velocity limit 
		tEnableDelay	: TIME 	:= T#0MS	;
		tDisableDelay	: TIME 	:= T#500MS  ;
	// ==== Axis data ====
		fEncoderTurnoverValue	: LREAL ;   
		
END_VAR
VAR // Axis configuration 
	// ===== HW Config Bits =====
		bIcfCmdVelocityRpm	: BOOL ; // input speeds in Rpm
		bIcfEnableForward 	: BOOL ; // Enable forward motion
 		bIcfEnablereverse	: BOOL ; // Enable reverse motion
		bIcfAlwaysEnable	: BOOL ; // 1 = Axis always enabled, 0 = Axis disabled at Idle 
		bIcfSimulationMode	: BOOL := FALSE ; // Simulation mode is active [default set to False] 
		bIcfModuloAxis		: BOOL := FALSE ; // Show axis position as modulo
		bIcfSTOPresent		: BOOL := FALSE ; // Axis Safe torque off is present
		bIcfNCHomeSensor	: BOOL := FALSE ; // Homing sensor is inverted (NC)	
	// ===== Internal motion values ======
		fHomePosition		: LREAL := 0 ; // set position at homing
	// Command Modes
		mcHomingMode 		: MC_HomingMode := MC_direct ; // Homing Mode ( MC_DefaultHoming, MC_Direct, MC_ForceCallibration, MC_ResetCallibration)
	// Values from system
		McReadSysVelo		: MC_ReadParameter		; // Read Acceleration parameter from drive 
		McReadSysAcc		: MC_ReadParameter		; // Read Acceleration parameter from drive 
		McReadSysDec		: MC_ReadParameter		; // Read Acceleration parameter from drive 
END_VAR
VAR	// ====== Axis enable =====
		bCmdEnableAxis 		: BOOL 	:= FALSE; // Command to enable the axis (External)
		bInternalEnable		: BOOL 	:= FALSE; // internal enable command (turns off after set time, and on at new motion command
		bAxisIsEnabled		: BOOL 	:= false; // Axis is enabled and ready for commands
		bDelayedEnable		: BOOL 	:= false; // Delayed enable signal for motion commands
		TonMotionEnable		: TON 			; // Timer on for motion command enable
		TofIntAxisEnable	: TOF  			; // Timer off for internal axis enable 
		bSTOOK				: BOOL 	:= FALSE; // Axis safet torque off is ok
		{attribute 'analysis' := '-33'}
		reSTOOK				: R_TRIG		; // rising edge safe torcue off ok
		tonSTOOK			: TON	; // Safe torque off ok timer
	// Parameter read status 
		Cmd_EnDriveParRead	: BOOL 			; // Enable parameter read 
	// ===== Physical Homing signal =====
		IAxisHome 	AT %I* 	: BOOL 			; // Axis homing sensor from PLC (if MC_DefaultHoming is used)
		IAxisSTOOK	AT %I* 	: BOOL 			; // Axis STO is ok
END_VAR
VAR	// =============== Motion status functions ================
	// =============== Motion function blocks =================
		fbMcPower 			: MC_Power		;		// FB for enable and override
		fbMcReset 			: MC_Reset		;		// FB to reset axis
		fbSoeReset			: FB_SoEReset	; 		// FB to reset axis hardware
		fbMcHome			: MC_Home		;		// Fb to home Axis
		fbMcStop 			: MC_Stop		;		// FB to stop axis
		fbMcHalt			: MC_Halt		;		// FB to halt axis
		fbMcJog				: MC_Jog		;		// FB to Jog axis
		fbMcMoveVelocity	: MC_MoveVelocity;		// FB to move with specified velocity until Next command is given
		fbMcGearInSlave		: MC_GearIn		;		// FB to gear axis to master 
		fbMcGearInDyn		: MC_GearInDyn	;		// FB to gear axis dynamicly to master
		fbMcGearOutSlave	: MC_GearOut	;		// FB to decouple gearing
		fbMcSetPosition		: MC_SetPosition;		// FB to Set axis position
//		fbMcWriteParameter	: MC_WriteParameterPersistent ; // FB to write parameters in persistend data

	(* PtoP Motion move commands are in arrays so multiple commands can be stacked *) 
		fbMCMoveRelative	: ARRAY [0..1] OF MC_MoveRelative	;		// FB to move relative
		fbMcMoveAbsolute	: ARRAY [0..1] OF MC_MoveAbsolute	;		// FB to move axis (velocity movement)
		fbMcMoveModulo		: ARRAY [0..1] OF MC_MoveModulo		;		// FB to move axis to modulo position
	// ===== Safe commands =====
		bCmdSafeStop		: BOOL ;
		bCmdSafeSpeed		: BOOL ; 
	// ===== Function execute triggers =====
		bExec_Reset			: BOOL := FALSE; // Execute reset
		bExec_Halt			: BOOL := FALSE; // Execute hold
		bExec_Home			: BOOL := FALSE; // Execute Home
		bExec_JogPositive	: BOOL := FALSE; // Execute Jog in positive direction
		bExec_JogNegative	: BOOL := FALSE; // Execute Jog in negative direction
		bExec_MoveVelocity	: BOOL := FALSE; // Execute move velocity
		bExec_GearAsSlave	: BOOL := FALSE; // Execute gear as slave
		bExec_GearSlaveDyn	: BOOL := FALSE; // Execute gear slave dynamic
		bExec_GearOutSlave	: BOOL := FALSE; // Execute gear out slave
		bExec_SetPosition	: BOOL := FALSE; // execute set position
//		bExec_ParWritePers	: BOOL := FALSE; // Execute parameter write persistent 
		
	(* PtoP Motion move commands are in arrays so multiple commands can be stacked *) 
		arExec_MoveRelative	: ARRAY [0..1] OF BOOL ; // Execute move relative
		arExec_MoveAbs		: ARRAY [0..1] OF BOOL ; // Execute move absolute reverse
		arExec_MoveModulo	: ARRAY [0..1] OF BOOL ; // Execute move modulo

		tonResetDone		: TON := (PT := T#300MS) ;
//		bCmd_MoveRelative	: BOOL		; // Move relative command
//		bCmd_MoveAbs		: BOOL		; // Move relative command
//		bCmd_MoveModulo		: BOOL		; // Move relative command
	
//		ReCmd_MoveRelative	: R_TRIG	; // Move Relative comamnd trigger
//		ReCmd_MoveAbs		: R_TRIG	; // Move Absolute comamnd trigger
//		ReCmd_MoveModulo	: R_TRIG	; // Move Modulo comamnd trigger

	// ===== Move ristrictions ======
		bCmdLimitVelocity 	: BOOL := FALSE			; // velocity limiting is active 
		fCmdVelocityLimit	: LREAL:= 100			; // Maximum velocity limit when velocity limiting is active  
		fSafeOverride		: LREAL:= 10 			; // [%] Safe velocity override  
		
	// ===== Internal variables =======
		fAcceleration		: LREAL := 0 ; // Acceleration used for functions 
		fDeceleration		: LREAL := 0 ; // Deceleration used for functions
		{attribute 'analysis' := '-33'}
		reCmdReset			: R_TRIG ; // Rising edge on reset command
END_VAR
VAR
	// ===== Loop variables =====
		i : DINT := 0 ; // For loop increment
	// ===== check variable ======
		rtrigInPosition	: R_TRIG ; // in position trigger
	// ===== Par write timer ===== 
END_VAR
VAR // Parameters 
	ParAccManualScaling	: Udt_Parameter := (fValue := 50, fFactory := 50, bTeachable := FALSE)  ; // Acceleration scaling factor for manual functions 
	ParDecManualScaling	: Udt_Parameter := (fValue := 50, fFactory := 50, bTeachable := FALSE)	; // Deceleration scaling factor for manual functions 
END_VAR

// Call base function
SUPER^(refFbFault := refFbFault);

// ==== Check if axis is initiated =====
IF NOT bInitOk THEN 
	RETURN ; 
END_IF
// ===== Execute safe functions =====
	ExecSafeFunctions(); 
	
// ==== Execute organizational functions =====
	CallOrganizationFunctions();
// ==== execute motion functions =====
	CallMotionFunctions();

METHOD PRIVATE CallMotionFunctions : BOOL
VAR_INPUT
END_VAR
// ===== Set acceleratio and deceleration values =======
	IF bCmdManual THEN 
		fAcceleration 	:= fCmdAcc * (ParAccManualScaling.fvalue / 100);
		fDeceleration	:= fCmdDecc* (ParDecManualScaling.fValue / 100);
	END_IF

// ===== block all other commands if axis is coupled =====
	IF NOT AxisRef.Status.Coupled THEN 
	// ===== Homing functions =====
		ExecHome		(); 
	
	// ===== Motion standstil commands =====
		ExecHalt		();
	
	// ===== Motion move functions
		ExecJog			();
		ExecMoveAbsolute();
		ExecMoveRelative();
		ExecMoveModulo	();
		ExecMoveVelocity();
	END_IF
	
// ===== Execute gearing functions =====
	ExecGearOut		();
	ExecGearIn		();
	ExecGearDynamic	();
	
// ====== reset velocity lmiting =====
	bVelocityLimited	:= bCmdLimitVelocity ;	
	bCmdLimitVelocity 	:= FALSE ; 

// ====== Reset acceleration deceleration values ======
	fAcceleration	:= fCmdAcc;
	fDeceleration	:= fCmdDecc;
END_METHOD

METHOD PRIVATE CallOrganizationFunctions : BOOL
VAR_INPUT
END_VAR
// ==== execute organizational functions =====
	ExecReadStatus		(); 
	ExecEnable			();
	ExecReset			();
//	ExecWriteParameter	();
	ExecSetPosition		();
END_METHOD

METHOD PUBLIC CmdGearDynamic : BOOL // Set axis to geared, activates with variable gear ratio until geared out or stopped (if method is no longer called then gear ratio is locked to last value)
VAR_INPUT
	fGearRatio	:	LREAL	:= 1	; // Slave Axis gearing ratio (Master = 1/ fGearRatio = Slave)	
END_VAR
// set blocked command if halt is active 
bBlockedCommand 		:= fbMcHalt.Active ;

// check if command buffer is empty 
	IF AxisRef.Status.CmdBuffered THEN 
		RETURN ;
	END_IF 

// Set command to true 
	bExec_GearSlaveDyn 	:= TRUE ;
	bInternalEnable		:= TRUE ;

// coppy parameters
	fCmdGearRatio 		:= fGearRatio ;

// Set feedback output 
	CmdGearDynamic 		:= bGearedAsSlave ;
END_METHOD

METHOD PUBLIC CmdGearIn : BOOL // Set axis to geared, activates with constant gear ratio until geared out or stopped
VAR_INPUT
	fGearRatio	:	LREAL	:= 1	; // Slave Axis gearing ratio (Master = 1/ fGearRatio = Slave)	
END_VAR
// set blocked command if halt is active 
	bBlockedCommand := fbMcHalt.Active ;

// check if command buffer is empty 
	IF AxisRef.Status.CmdBuffered THEN 
		RETURN ;
	END_IF 
	
// Set command to true 
	bExec_GearAsSlave 	:= TRUE ;
	bInternalEnable		:= TRUE ;

// coppy parameters
	fCmdGearRatio 				:= fGearRatio ;

// Set feedback output 
	CmdGearIn := bGearedAsSlave ;
END_METHOD

METHOD CmdGearOut : BOOL
VAR_INPUT
END_VAR
// set blocked command if halt is active 
bBlockedCommand := fbMcHalt.Active ;

// Set command to true
bExec_GearOutSlave 	:= TRUE ;
bExec_GearAsSlave	:= FALSE;
bExec_GearSlaveDyn 	:= FALSE;

// Set feedback Output
CmdGearOut := fbMcGearOutSlave.Done;
END_METHOD

METHOD PUBLIC CmdHalt : BOOL
VAR_INPUT
	fDeceleration 	: LREAL := 0 ; // command deceleration
	mcBuffermode	: MC_BufferMode ; // Buffermode defines how the previous command is executed.
END_VAR
// Set command to true 
bExec_Halt 		:= TRUE ;
bInternalEnable	:= TRUE ;

// coppy parameters
fbMcHalt.Deceleration	:= fDeceleration;
fbMcHalt.BufferMode		:= mcBuffermode	;

// Set feedback output 
CmdHalt := fbMchalt.Active OR fbMcHalt.Done ;
END_METHOD

METHOD PUBLIC CmdHold : BOOL
VAR_INPUT
END_VAR
// Set command to true 
bExec_Halt 		:= TRUE ;
bInternalEnable	:= TRUE ;

// coppy parameters
fbMcHalt.Deceleration	:= 0;
fbMcHalt.BufferMode		:= 0;

// Set feedback output 
CmdHold := fbMchalt.Active OR fbMcHalt.Done ;
END_METHOD

METHOD PUBLIC CmdHome : BOOL // start axis homing procedure
VAR_INPUT
	fPosition 		: LREAL := 0 ; // Homing position
END_VAR
// set blocked command if halt is active 
bBlockedCommand := fbMcHalt.Active ;

// set command to true 
bExec_Home 		:= TRUE	; 
bInternalEnable	:= TRUE ;

// coppy parameters
fbMcHome.Position 	:= fPosition 	;

// Set feedback output
CmdHome := fbMcHome.Done ;
END_METHOD

METHOD PUBLIC CmdJog : BOOL // Jog axis with variable speed. jog stops as soon as the command is false
VAR_INPUT
	fVelocity		: LREAL 	; // jog velocity can be adjusted as long as the command is active
	fPos			: LREAL 	; // Jog position or step size (if aplicable)
	bJogNegative 	: BOOL 		:= FALSE ; // jog in negative direction
	eJogmode		: E_JogMode := E_JogMode.MC_JOGMODE_CONTINOUS ; // jogmode [default MC_JOGMODE_CONTINOUS] 
END_VAR
// set blocked command if halt is active 
bBlockedCommand := fbMcHalt.Active ;

// Velocity conversion from RPM to deg/sec
	IF bIcfCmdVelocityRpm THEN 
		fVelocity := Rpm_To_DegS(fVelocity);
	END_IF

// Set command to true
	IF fbMcJog.Velocity = fVelocity THEN // If command velocity changes, then set exec to false for one cycle to trigger new velocity so the jog follows the set velocity
		bExec_JogPositive	:= NOT bJogNegative ;
		bExec_JogNegative 	:= bJogNegative ;
	END_IF
	bInternalEnable			:= TRUE ;

// coppy parameters
	fbMcJog.Velocity	:= fVelocity 	;
	fbmcjog.Mode		:= eJogmode		;
	fbMcJog.Position	:= fPos			;

// Set feedback output 
	CmdJog := fbMcJog.Active ;
END_METHOD

METHOD PUBLIC CmdKeepEnabled : BOOL
VAR_INPUT
END_VAR
// Keep internal enable on while command is active
bInternalEnable			:= TRUE ;
END_METHOD

METHOD PUBLIC CmdLimitVelocity : BOOL // limit axis maximum velocity, stays active as long as command is called. 
VAR_INPUT
	fVelocityLimit	: LREAL ; // velocity Maximum limit
END_VAR
// set blocked command if halt is active 
bBlockedCommand := fbMcHalt.Active ;

// Set velocity limiting command 
bCmdLimitVelocity S= TRUE;
	
// Set velocity maximum value 
fCmdVelocityLimit := fVelocityLimit ; 

// set feedback 
CmdLimitVelocity := bVelocityLimited ;
END_METHOD

METHOD PUBLIC CmdManual : BOOL
VAR
	eJogmode		: E_JogMode := E_JogMode.MC_JOGMODE_CONTINOUS ; // jogging mode 
END_VAR
// set blocked command if halt is active 
bBlockedCommand := fbMcHalt.Active ;

// Enable axis for manual control
bCmdManual := TRUE ;

// check safety 
IF NOT bSafetyOk THEN 
	RETURN;
END_IF

// set jog mode 
IF stManualCtrl.bCmdInching THEN 
	eJogmode := E_JogMode.MC_JOGMODE_INCHING ;
END_IF

// execute motion commands
IF stManualCtrl.bCmdJogForward OR stManualCtrl.bCmdJogReverse THEN 
	CmdJog (fVelocity := stManualCtrl.fVelocity, 
			fPos := stManualCtrl.fDistance, 
			bJogNegative := stManualCtrl.bCmdJogReverse, 
			eJogmode := eJogmode);
ELSIF stManualCtrl.bCmdToPos THEN 
	CmdMoveAbs( fPosition := stManualCtrl.fPosition, 
				fVelocity := stManualCtrl.fVelocity, 
				mcBuffermode := MC_BufferMode.MC_Aborting);
ELSIF stManualCtrl.bCmdHome THEN 
	CmdHome( fPosition := 0);
ELSE 
	CmdHalt( 	fDeceleration := fMaxDec * 0.9, 
				mcBuffermode := MC_BufferMode.MC_Aborting) ; 
END_IF
END_METHOD

METHOD PUBLIC CmdMoveAbs : BOOL // Move absolute command
VAR_INPUT
	fPosition	:	LREAL 	; // target position
	fVelocity	: 	LREAL 	; // Maximum velocity [units/sec]
	mcBuffermode: 	MC_BufferMode ; // Buffermode defines how the previous command is executed.
END_VAR
// set blocked command if halt is active 
bBlockedCommand := fbMcHalt.Active ;

// Velocity conversion from RPM to deg/sec
	IF bIcfCmdVelocityRpm THEN 
		fVelocity := Rpm_To_DegS(fVelocity);
	END_IF

// Determine function for command stacking
IF NOT AxisRef.Status.CmdBuffered OR mcBuffermode <> MC_Aborting THEN 
	IF fbMcMoveAbsolute[0].Active THEN 
		arExec_MoveAbs[1] 				:= (fPosition <> fbMcMoveAbsolute[0].Position OR fVelocity <> fbMcMoveAbsolute[0].Velocity) ;
		fbMcMoveAbsolute[1].Position 	:= fPosition ;
		fbMcMoveAbsolute[1].Velocity 	:= fVelocity ; 
		fbMcMoveAbsolute[1].BufferMode 	:= mcBuffermode ;
	ELSE
		arExec_MoveAbs[0] 				:= (fPosition <> fbMcMoveAbsolute[1].Position OR fVelocity <> fbMcMoveAbsolute[1].Velocity) ;
		fbMcMoveAbsolute[0].Position 	:= fPosition ;
		fbMcMoveAbsolute[0].Velocity 	:= fVelocity ; 
		fbMcMoveAbsolute[0].BufferMode 	:= mcBuffermode ;
	END_IF
END_IF
	
bInternalEnable	:= TRUE ;

// set feedback
IF arExec_MoveAbs[1] OR fbMcMoveAbsolute[1].Busy THEN 
	CmdMoveAbs :=	fbMcMoveAbsolute[1].Active ;
ELSE 
	CmdMoveAbs :=	fbMcMoveAbsolute[0].Active ;
END_IF
END_METHOD

METHOD PUBLIC CmdMoveModulo : BOOL // Move to a modulo position
VAR_INPUT
	fPosition	:	LREAL 	; // target position
	fVelocity	: 	LREAL 	; // Maximum velocity [units/sec]
	mcDirection : 	MC_Direction := MC_Direction.MC_Positive_Direction ; // Direction of movement mc_direction [ deafult mc_positive_direction]
	mcBuffermode: 	MC_BufferMode ; // Buffermode defines how the previous command is executed.
END_VAR
// set blocked command if halt is active 
bBlockedCommand := fbMcHalt.Active ;


// Velocity conversion from RPM to deg/sec
	IF bIcfCmdVelocityRpm THEN 
		fVelocity := Rpm_To_DegS(fVelocity);
	END_IF

// Determine function for command stacking
IF NOT AxisRef.Status.CmdBuffered OR mcBuffermode <> MC_Aborting THEN 
	IF fbMcMoveModulo[0].Busy THEN 
		arExec_MoveModulo[1] 		:= (fPosition <> fbMcMoveModulo[0].Position OR fVelocity <> fbMcMoveModulo[0].Velocity)	;
		fbMcMoveModulo[1].Velocity 	:= fVelocity 	;
		fbMcMoveModulo[1].Position 	:= fPosition 	;
		fbMcMoveModulo[1].Direction	:= mcDirection	;
		fbMcMoveModulo[1].BufferMode:= mcBuffermode ;
	ELSE    
		arExec_MoveModulo[0] 		:= (fPosition <> fbMcMoveModulo[1].Position OR fVelocity <> fbMcMoveModulo[1].Velocity) ;
		fbMcMoveModulo[0].Velocity 	:= fVelocity 	;
		fbMcMoveModulo[0].Position 	:= fPosition 	;
		fbMcMoveModulo[0].Direction	:= mcDirection	;
		fbMcMoveModulo[0].BufferMode:= mcBuffermode ;
	END_IF
END_IF 
	
bInternalEnable	:= TRUE ;

// set feedback
IF arExec_MoveModulo[1] OR fbMcMoveModulo[1].Busy THEN 
	CmdMoveModulo :=	fbMcMoveModulo[1].Active OR fbMcMoveModulo[1].Done;
ELSE
	CmdMoveModulo :=	fbMcMoveModulo[0].Active OR fbMcMoveModulo[0].Done ;
END_IF
END_METHOD

METHOD CmdMoveRelative : BOOL // move relative command 
VAR_INPUT
	fDistance	:	LREAL 	; // target position
	fVelocity	: 	LREAL 	; // Maximum velocity [units/sec]
	mcBuffermode: 	MC_BufferMode ; // Buffermode defines how the previous command is executed.
END_VAR
// set blocked command if halt is active 
bBlockedCommand := fbMcHalt.Active ;

// Velocity conversion from RPM to deg/sec
	IF bIcfCmdVelocityRpm THEN 
		fVelocity := Rpm_To_DegS(fVelocity);
	END_IF

// Determine function for command stacking
IF NOT AxisRef.Status.CmdBuffered OR mcBuffermode <> MC_Aborting THEN 
	IF fbMCMoveRelative[0].Active THEN 
		arExec_MoveRelative[1] := (fDistance <> fbMCMoveRelative[0].Distance OR fVelocity <> fbMCMoveRelative[0].Velocity) ;
		fbMCMoveRelative[1].Velocity	:= fVelocity 	;
		fbMCMoveRelative[1].Distance	:= fDistance	;
		fbMCMoveRelative[1].BufferMode	:= mcBuffermode	;
	ELSE 
		arExec_MoveRelative[0] := (fDistance <> fbMCMoveRelative[1].Distance OR fVelocity <> fbMCMoveRelative[1].Velocity) ;
		fbMCMoveRelative[0].Velocity	:= fVelocity 	;
		fbMCMoveRelative[0].Distance	:= fDistance	;
		fbMCMoveRelative[0].BufferMode	:= mcBuffermode	;
	END_IF
END_IF
bInternalEnable	:= TRUE ;

// set feedback
IF arExec_MoveRelative[1] OR fbMCMoveRelative[1].Busy THEN 
	CmdMoveRelative :=	fbMCMoveRelative[1].Active ;
ELSE
	CmdMoveRelative :=	fbMCMoveRelative[0].Active ;
END_IF
END_METHOD

METHOD PUBLIC CmdMoveVelocity : BOOL // Move with set velocity until stopped
VAR_INPUT
	fVelocity	: 	LREAL 	; // Maximum velocity [units/sec]
	mcDirection : 	MC_Direction := MC_Direction.MC_Positive_Direction ; // Direction of movement mc_direction [ deafult mc_positive_direction]
	mcBuffermode: 	MC_BufferMode ; // Buffermode defines how the previous command is executed.
END_VAR
// set blocked command if halt is active 
bBlockedCommand := fbMcHalt.Active ;

// Velocity conversion from RPM to deg/sec
	IF bIcfCmdVelocityRpm THEN 
		fVelocity := Rpm_To_DegS(fVelocity);
	END_IF

// Set command to true 
	IF NOT AxisRef.Status.CmdBuffered OR mcBuffermode <> MC_Aborting THEN 
		bExec_MoveVelocity 	:= TRUE ;
		bInternalEnable		:= TRUE ;
	END_IF
	
// coppy parameters
	fbMcMoveVelocity.Velocity	:= fVelocity 	;
	fbMcMoveVelocity.Direction 	:= mcDirection	;
	fbMcMoveVelocity.BufferMode	:= mcBuffermode	;

// Set feedback output 
	CmdMoveVelocity := fbMcMoveVelocity.Active ;
END_METHOD

METHOD PUBLIC CmdOverwriteAcc : BOOL // temporarilly overwrite deceleration values
VAR_INPUT	
	fValue	: LREAL ; // Overwrite value 
END_VAR
fAcceleration := fValue ;

CmdOverwriteAcc := TRUE ;
END_METHOD

METHOD PUBLIC CmdOverwriteDec : BOOL // Temporarilly overwrite deceleration values
VAR_INPUT
	fValue	: LREAL ; // Overwrite value 
END_VAR
fDeceleration := fValue ;

CmdOverwriteDec := TRUE ;
END_METHOD

METHOD PUBLIC CmdReset : BOOL
VAR_INPUT
END_VAR
// Set reset axis to true 				
	bExec_Reset 	:= TRUE ; 
	bInternalEnable	:= TRUE ;
	
// Set feedback output 
	CmdReset := tonResetDone.Q ;
END_METHOD

METHOD PUBLIC CmdSafeSpeed : BOOL
VAR_INPUT
END_VAR
// Set safestop command
bCmdSafeSpeed := TRUE ; 

// Set feedback output 
CmdSafeSpeed := fbMcPower.Override = fSafeOverride  ;
END_METHOD

METHOD PUBLIC CmdSafeStop : BOOL
VAR_INPUT
END_VAR
IF AxisRef.Status.Coupled THEN 
	CmdSafeStop := AxisRef.Status.NotMoving ;
	RETURN;
END_IF
// Set safestop command
bCmdSafeStop := TRUE ; 

// Set feedback output 
CmdSafeStop := bIsSafe OR NOT bInitOk;
END_METHOD

METHOD PUBLIC CmdSetPosition : BOOL
VAR_INPUT
	fPosition		: LREAL ; // encoder position
	bSetRelative	: BOOL 	; // TRUE = relative position offset, FALSE = Absolute position
END_VAR
bExec_SetPosition 			:= NOT fbMcSetPosition.Busy AND NOT fbMcSetPosition.Done ; 
fbMcSetPosition.Position	:= fPosition ;
fbMcSetPosition.Mode		:= bSetRelative ;

CmdSetPosition := fbMcSetPosition.Done;
END_METHOD

METHOD PRIVATE ExecEnable : BOOL
VAR_INPUT
END_VAR
// ===== Set axis enable ======
IF NOT bSafetyOk 
OR NOT bSTOOK 
OR AxisRef.Status.DriveDeviceError
OR bExec_Reset THEN 
	bCmdEnableAxis := FALSE ;
ELSIF bCmdManual AND bSafetyOk THEN 
	bCmdEnableAxis 	:= TRUE ;
	bInternalEnable S= bCmdManual ;
	bCmdManual 		:= FALSE ;
ELSE 
	bCmdEnableAxis	:= bEnable ;
END_IF

// ===== Check if axis is bussy with a command =====
	bInternalEnable S= AxisRef.Status.HasJob;
	bInternalEnable	S= bIcfAlwaysEnable ; // always enable axis if configured
	bInternalEnable	S= AxisRef.Status.Coupled ;

// ===== Axis disable timer after last command =====
	TofIntAxisEnable (	IN:= bInternalEnable, PT := tDisableDelay);

// ===== Enable drive =====
	fbMcPower(	Axis			:= AxisRef , 
				Enable			:= bCmdEnableAxis AND TofIntAxisEnable.Q, 
				Enable_Positive	:= bIcfEnableForward, 
				Enable_Negative	:= bIcfEnablereverse, 
				BufferMode		:= MC_Buffered );  
				
// ===== Reset internal enable signal =====
	bInternalEnable := FALSE ; 	

// ===== Delayed enable function =====	
	IF fbMcPower.Enable AND fbMcPower.Status THEN
		bAxisIsEnabled := TRUE ;
	ELSIF NOT fbMcPower.Enable OR AxisRef.Status.Error THEN 
		bAxisIsEnabled := FALSE ; 
	END_IF

	TonMotionEnable	(IN := bAxisIsEnabled, PT := tEnableDelay);
	bDelayedEnable 	:= TonMotionEnable.Q ;	

IF AxisRef.Status.DriveDeviceError 
AND bCmdEnableAxis THEN
	bError					:= TRUE							;
	stFault.Active 			:= TRUE 						;
	stFault.MessageNumber	:= E_MessageNumbers.FF_AxisFault;
	stFault.Discription		:= CONCAT('Drive device error ', UDINT_TO_STRING(AxisRef.Status.ErrorID));
	stFault.Discription		:= CONCAT( sName , stfault.Discription ) ;
	stFault.FaultType		:= E_FaultTypes.FF				;
ELSIF fbMcPower.Error THEN 
	bError					:= TRUE							;
	stFault.Active 			:= TRUE 						;
	stFault.MessageNumber	:= E_MessageNumbers.FF_AxisFault;
	stFault.Discription		:= CONCAT('Enable Fault ', UDINT_TO_STRING(fbMcPower.ErrorID));
	stFault.Discription		:= CONCAT( sName , stfault.Discription ) ;
	stFault.FaultType		:= E_FaultTypes.FF				;
END_IF
END_METHOD

METHOD INTERNAL ExecGearDynamic : BOOL
VAR_INPUT
END_VAR
// ===== invert gear ratio if reverse slave is active =====
	IF bReverseSlave THEN 
		fbMcGearInDyn.GearRatio := fCmdGearRatio * -1 ;
	ELSE 
		fbMcGearInDyn.GearRatio := fCmdGearRatio ;
	END_IF

// ===== Execute gear in function =====
	fbMcGearInDyn ( 	Master 			:= refMasterAxis,
						Slave			:= AxisRef,
						Enable 			:= bExec_GearSlaveDyn AND bDelayedEnable,
						Acceleration	:= 0,
						Deceleration	:= 0	); 
						
// ===== reset command =====
	bExec_GearSlaveDyn	:= FALSE ;
	bGearedAsSlave		:= fbMcGearInDyn.InGear ; 

// Gearing fault handling 
	IF fbMcGearInDyn.Error THEN 
		bError					:= TRUE							;
		stFault.Active 			:= TRUE 						;
		stFault.MessageNumber	:= E_MessageNumbers.FF_AxisFault;
		stFault.Discription		:= CONCAT('Gear dynamic Fault ', UDINT_TO_STRING(fbMcGearInDyn.ErrorID));	
		stFault.Discription		:= CONCAT( sName , stfault.Discription ) ;
		stFault.FaultType		:= E_FaultTypes.FF				;
	END_IF
END_METHOD

METHOD INTERNAL ExecGearIn : BOOL
VAR_INPUT
END_VAR
// ===== invert gear ratio if reverse slave is active =====
	IF bReverseSlave THEN 
		fbMcGearInSlave.RatioNumerator := fCmdGearRatio * -1 ;
	ELSE 
		fbMcGearInSlave.RatioNumerator := fCmdGearRatio ;
	END_IF

// ===== Execute gear in function =====
	fbMcGearInSlave ( 	Master 			:= refMasterAxis,
						Slave			:= AxisRef,
						Execute 		:= bExec_GearAsSlave AND bDelayedEnable,
						RatioDenominator:= 1,
						Acceleration	:= 0,
						Deceleration	:= 0	); 
						
// ===== reset command =====
	bExec_GearAsSlave 	:= FALSE  ;
	bGearedAsSlave		S= fbMcGearInSlave.InGear ; 

// Gearing fault handling 
	IF fbMcGearInSlave.Error THEN 
		bError					:= TRUE							;
		stFault.Active 			:= TRUE 						;
		stFault.MessageNumber	:= E_MessageNumbers.FF_AxisFault;
		stFault.Discription		:= CONCAT('Gear as slave Fault ', UDINT_TO_STRING(fbMcGearInSlave.ErrorID));
		stFault.Discription		:= CONCAT( sName , stfault.Discription ) ;
		stFault.FaultType		:= E_FaultTypes.FF				;
	END_IF
END_METHOD

METHOD INTERNAL ExecGearOut : BOOL
VAR_INPUT
END_VAR
// ===== execute gear out function ======
	fbMcGearOutSlave (	Slave 	:= AxisRef,
						Execute := bExec_GearOutSlave );

// ===== reset command =====
	bExec_GearOutSlave	:= false ;
	bGearedAsSlave		R= fbMcGearOutSlave.Done 	; 

// Gearing fault handling 
	IF fbMcGearOutSlave.Error THEN 
		bError					:= TRUE							;
		stFault.Active 			:= TRUE 						;
		stFault.MessageNumber	:= E_MessageNumbers.FF_AxisFault;
		stFault.Discription		:= CONCAT('Gear out Fault ', UDINT_TO_STRING(fbMcGearOutSlave.ErrorID));
		stFault.Discription		:= CONCAT( sName , stfault.Discription ) ;
		stFault.FaultType		:= E_FaultTypes.FF				;
	END_IF
END_METHOD

METHOD INTERNAL ExecHalt : BOOL
VAR_INPUT
END_VAR
// ==== Execute halt function ===== 
fbMcHalt (	Axis 		:= AxisRef,
			Execute 	:= bExec_Halt );

// ===== reset command =====
	bExec_Halt := FALSE ;
	
// Halt fault handling 
	IF fbMcHalt.Error THEN 
		bError					:= TRUE							;
		stFault.Active 			:= TRUE 						;
		stFault.MessageNumber	:= E_MessageNumbers.FF_AxisFault;
		stFault.Discription		:= CONCAT('Halt Fault ', UDINT_TO_STRING(fbMcHalt.ErrorID));
		stFault.Discription		:= CONCAT( sName , stfault.Discription ) ;
		stFault.FaultType		:= E_FaultTypes.FF				;
	END_IF
END_METHOD

METHOD INTERNAL ExecHome : BOOL
VAR_INPUT
END_VAR
// ==== execute homing function =====
	IF bIcfNCHomeSensor THEN 
		fbmchome.bCalibrationCam	:= NOT IAxisHome;
	ELSE
		fbmchome.bCalibrationCam	:= IAxisHome;
	END_IF		
		
	fbMcHome(	Axis			:= AxisRef,
				Execute			:= bExec_Home AND bDelayedEnable,
				HomingMode		:= mcHomingMode ); 
			
// Reset exec command 
	bExec_Home 	:= FALSE ;
	bHomed		S= fbMcHome.Done ;	
				
// fault handling 
	IF fbMcHome.Error THEN 
		bError					:= TRUE							;
		stFault.Active 			:= TRUE 						;
		stFault.MessageNumber	:= E_MessageNumbers.FF_AxisFault;
		stFault.Discription		:= CONCAT('Homing Fault ', UDINT_TO_STRING(fbMcHome.ErrorID));
		stFault.Discription		:= CONCAT( sName , stfault.Discription ) ;
		stFault.FaultType		:= E_FaultTypes.FF				;
	END_IF
END_METHOD

METHOD INTERNAL ExecJog : BOOL
VAR_INPUT
END_VAR
// ===== Execute Jog function =====
	IF bCmdLimitVelocity THEN 
		fbMcJog.Velocity := MIN(fCmdVelocityLimit, fbMcJog.Velocity); 
	END_IF

	// function call
	fbMcJog (	Axis 		:= AxisRef,
				JogForward	:= bExec_JogPositive AND bDelayedEnable,
				JogBackwards:= bExec_JogNegative AND bDelayedEnable,
				Acceleration:= fAcceleration,
				Deceleration:= fDeceleration );

// ===== reset command =====
	bExec_JogPositive 	:= FALSE  ;
	bExec_JogNegative	:= FALSE  ;
	
// Jog fault handling 
	IF fbMcJog.Error THEN 
		bError					:= TRUE							;
		stFault.Active 			:= TRUE 						;
		stFault.MessageNumber	:= E_MessageNumbers.FF_AxisFault;
		stFault.Discription		:= CONCAT('Jog Fault ', UDINT_TO_STRING(fbMcJog.ErrorID));
		stFault.Discription		:= CONCAT( sName , stfault.Discription ) ;
		stFault.FaultType		:= E_FaultTypes.FF				;
	END_IF
END_METHOD

METHOD INTERNAL ExecMoveAbsolute : BOOL
VAR_INPUT
END_VAR
// ==== execute move absolute function =====
FOR i := 0 TO 1 DO 
	// Limit velocity
	IF bCmdLimitVelocity THEN 
		fbMcJog.Velocity := MIN(fCmdVelocityLimit, fbMcMoveAbsolute[i].Velocity); 
	END_IF
	// function call
	fbMcMoveAbsolute[i](	Axis 		:= AxisRef,
							Execute 	:= arExec_MoveAbs[i] AND bDelayedEnable,
							Acceleration:= fAcceleration,
							Deceleration:= fDeceleration );  

	// If function is done then reset command values
	IF fbMcMoveAbsolute[i].Done OR fbMcMoveAbsolute[i].CommandAborted OR NOT arExec_MoveAbs[i] THEN 
		fbMcMoveAbsolute[i].Velocity	:= 0 ;
		fbMcMoveAbsolute[i].Position	:= 0 ; 
	END_IF

	// reset Exec command 
	arExec_MoveAbs[i] := FALSE ; 
	
	// fault handling 
	IF fbMcMoveAbsolute[i].Error THEN 
		bError					:= TRUE							;
		stFault.Active 			:= TRUE 						;
		stFault.MessageNumber	:= E_MessageNumbers.FF_AxisFault;
		stFault.Discription		:= CONCAT('Move absolute Fault ', UDINT_TO_STRING(fbMcMoveAbsolute[i].ErrorID));
		stFault.Discription		:= CONCAT( sName , stfault.Discription ) ;
		stFault.FaultType		:= E_FaultTypes.FF				;
	END_IF
END_FOR
END_METHOD

METHOD INTERNAL ExecMoveModulo : BOOL
VAR_INPUT
END_VAR


// ===== Execute move modulo function =====
FOR i := 0 TO 1 DO 
	IF bCmdLimitVelocity THEN 
		fbMcJog.Velocity := MIN(fCmdVelocityLimit, fbMcMoveModulo[i].Velocity); 
	END_IF
	// function call
	fbMcMoveModulo[i](	Axis 		:= AxisRef,
						Execute 	:= arExec_MoveModulo[i] AND bDelayedEnable,
						Acceleration:= fAcceleration,
						Deceleration:= fDeceleration);  
	
	// If function is done then reset command values
	IF fbMcMoveModulo[i].Done OR fbMcMoveModulo[i].CommandAborted OR NOT arExec_MoveModulo[i] THEN 
		fbMcMoveModulo[i].Velocity	:= 0 ;
		fbMcMoveModulo[i].Position	:= 0 ; 
	END_IF

	// reset Exec command 
	arExec_MoveModulo[i] := FALSE ; 
	
	// fault handling 
	IF fbMcMoveModulo[i].Error THEN 
		bError					:= TRUE							;
		stFault.Active 			:= TRUE 						;
		stFault.MessageNumber	:= E_MessageNumbers.FF_AxisFault;
		stFault.Discription		:= CONCAT('Move module Fault ', UDINT_TO_STRING(fbMcMoveModulo[i].ErrorID));
		stFault.Discription		:= CONCAT( sName , stfault.Discription ) ;
		stFault.FaultType		:= E_FaultTypes.FF			;
	END_IF
END_FOR
END_METHOD

METHOD INTERNAL ExecMoveRelative : BOOL
VAR_INPUT
END_VAR
//ReCmd_MoveModulo(CLK := bCmd_MoveModulo );
//bCmd_MoveModulo	:= FALSE ;

// ===== Execute move relative function ======
FOR i := 0 TO 1 DO 
	// Limit velocity
	IF bCmdLimitVelocity THEN 
		fbMcJog.Velocity := MIN(fCmdVelocityLimit, fbMcMoveModulo[i].Velocity); 
	END_IF
	// function call
	fbMCMoveRelative[i](	Axis 		:= AxisRef,
							Execute		:= arExec_MoveRelative[i] AND bDelayedEnable,
							Acceleration:= fAcceleration,
							Deceleration:= fDeceleration );

	// If function is done then reset command values
	IF fbMCMoveRelative[i].Done OR fbMCMoveRelative[i].CommandAborted OR NOT arExec_MoveRelative[i] THEN 
		fbMCMoveRelative[i].Velocity	:= 0 ;
		fbMCMoveRelative[i].Distance	:= 0 ; 
	END_IF

	// reset Exec command 
	arExec_MoveRelative[i] := FALSE ; 
	
	// fault handling 
	IF fbMCMoveRelative[i].Error THEN 
		bError					:= TRUE							;
		stFault.Active 			:= TRUE 						;
		stFault.MessageNumber	:= E_MessageNumbers.FF_AxisFault;
		stFault.Discription		:= CONCAT('Move relative Fault ', UDINT_TO_STRING(fbMCMoveRelative[i].ErrorID));
		stFault.Discription		:= CONCAT( sName , stfault.Discription ) ;
		stFault.FaultType		:= E_FaultTypes.FF			;
	END_IF
END_FOR
END_METHOD

METHOD INTERNAL ExecMoveVelocity : BOOL
VAR_INPUT
END_VAR
// ===== Execute move velocity function =====
	IF bCmdLimitVelocity THEN 
		fbMcJog.Velocity := MIN(fCmdVelocityLimit, fbMcMoveVelocity.Velocity); 
	END_IF

// function call
fbMcMoveVelocity (	Axis 		:= AxisRef,
					Execute		:= bExec_MoveVelocity  AND bDelayedEnable,
					Acceleration:= fAcceleration,
					Deceleration:= fDeceleration );

// ===== reset command =====
bExec_MoveVelocity := FALSE ;
	
// Halt fault handling 
IF fbMcMoveVelocity.Error THEN 
	bError					:= TRUE							;
	stFault.Active 			:= TRUE 						;
	stFault.MessageNumber	:= E_MessageNumbers.FF_AxisFault;
	stFault.Discription		:= CONCAT('Move velocity Fault ', UDINT_TO_STRING(fbMcMoveVelocity.ErrorID));
	stFault.Discription		:= CONCAT( sName , stfault.Discription ) ;
	stFault.FaultType		:= E_FaultTypes.FF				;
END_IF
END_METHOD

METHOD INTERNAL ExecReadStatus : BOOL
VAR_INPUT
END_VAR
AxisRef.ReadStatus();
					
// convert velocity to RPM for output if aplicable
IF bIcfCmdVelocityRpm THEN 
	fVelocity := AxisRef.NcToPlc.ActVelo / 6 ;
ELSE 
	fVelocity := AxisRef.NcToPlc.ActVelo ;
END_IF

// write position output
IF bIcfModuloAxis THEN 
	fActPosition := AxisRef.NcToPlc.ModuloActPos ;
ELSE
	fActPosition := AxisRef.NcToPlc.ActPos ;
END_IF
						
// set status bits 
bIdle := NOT AxisRef.Status.HasJob ;

// In position 
	rtrigInPosition( 	CLK := AxisRef.Status.InTargetPosition, 
						Q => bReInTargetPos);
END_METHOD

METHOD INTERNAL ExecReset : BOOL
VAR_INPUT
END_VAR
VAR
	xMcReset			: BOOL ; // Execute MC reset
	xSoeReset			: BOOL ; // Execute SOE reset

END_VAR
//IF  AxisRef.Status.Moving AND bExec_Reset THEN // If the axis is still moving execute safe stop first
//	RETURN;
IF AxisRef.Status.Coupled THEN 
	RETURN;
END_IF

// ===== reset command =====
	bError 		:= AxisRef.Status.Error ; 
	bExec_Reset	R= fbMcReset.Done  ;

// ==== execute reset functions =====
IF AxisRef.Status.DriveDeviceError AND IAxisSTOOK THEN 
		xSoeReset := TRUE ;
ELSIF bSTOOK AND bExec_Reset THEN
		xMcReset	:= TRUE ;
ELSE 
	xSoeReset 	:= FALSE ;
	xMcReset	:= FALSE ;
END_IF

fbSoeReset	( 	Execute := xSoeReset,
				Timeout	:= T#5S,
				Axis	:= AxisRef);

fbMcReset	( 	Execute	:= xMcReset,
				Axis	:= AxisRef ); 
				
// ===== Set feedback =====
	bResetDone 	S= fbMcReset.Done  ;
	bResetDone	R= AxisRef.Status.Error ;
	tonResetDone (IN	:= bResetDone);

// ===== reset limitations =====
	bCmdSafeSpeed 	:= FALSE ;

	
// Reset fault handling 
	IF fbSoeReset.Error OR fbMcReset.Error THEN 
		bError					:= TRUE							;
		stFault.Active 			:= TRUE 						;
		stFault.MessageNumber	:= E_MessageNumbers.FF_AxisFault;
		stFault.Discription		:= CONCAT('Reset Fault ', UDINT_TO_STRING(fbMcReset.ErrorID));
		stFault.Discription		:= CONCAT( sName , stfault.Discription ) ;
		stFault.FaultType		:= E_FaultTypes.FF				;
	END_IF
END_METHOD

METHOD PRIVATE ExecSafeFunctions : BOOL
VAR_INPUT
END_VAR
// ==== Stop when safety is not ok =====
	bCmdSafeStop S= NOT bSafetyOk ;

// ===== Safe torque off function =====
	IF bIcfSTOPresent THEN 
		tonSTOOK(IN := IAxisSTOOK, PT := T#1000MS);
		bSTOOK := tonSTOOK.Q AND NOT AxisRef.Status.DriveDeviceError;
//		bSTOOK	:= IAxisSTOOK ;
	ELSE 
		bSTOOK := true ;
	END_IF
	
// ==== Safe operation functions (overrule all other motion functions) =====
	IF NOT AxisRef.Status.Coupled AND bSTOOK THEN 
		fbMcStop( 	Axis 			:= AxisRef		,
					Execute 		:= bCmdSafeStop AND NOT bExec_Reset,
					Deceleration	:= fMaxDec		);
	END_IF
	
	// Reset axis command			
	bCmdSafeStop 	R= fbMcStop.Done OR AxisRef.Status.HasBeenStopped OR NOT bSTOOK ;
	bStopped		:= AxisRef.Status.HasBeenStopped OR NOT bSTOOK ;

// Safestop fault handling 
	IF fbMcStop.Error THEN 
		bError					:= TRUE							;
		stFault.Active 			:= TRUE 						;
		stFault.MessageNumber	:= E_MessageNumbers.FF_AxisFault;
		stFault.Discription		:= CONCAT('Safe stop axis fault ', UDINT_TO_STRING(fbMcStop.ErrorID));
		stFault.Discription		:= CONCAT( sName , stfault.Discription ) ;
		stFault.FaultType		:= E_FaultTypes.FF				;
	END_IF
	
// ===== Safe speed monitoring =====
	IF bCmdSafeSpeed THEN 
		fbMcPower.Override 	:= fSafeOverride ;
		bCmdSafeSpeed		:= FALSE ;
	ELSE 
		fbMcPower.Override := 100 ;
	END_IF

// ===== Dev is safe feedback =====
bIsSafe := AxisRef.Status.HasBeenStopped OR AxisRef.Status.Disabled  ;
END_METHOD

METHOD INTERNAL ExecSetPosition : BOOL
VAR_INPUT
END_VAR
// ====== set position of axis ======
IF bExec_SetPosition OR fbMcSetPosition.Busy THEN 
	fbMcSetPosition (	Axis 	:= AxisRef,
						Execute	:= bExec_SetPosition );
	bExec_SetPosition := TRUE ;
END_IF
END_METHOD

METHOD PRIVATE ExecWriteParameter : BOOL
VAR_INPUT
END_VAR
// check if axis is disabled before writeing parameter
	AxisRef.ReadStatus();
	IF AxisRef.Status.Disabled 
	AND (fbMcWriteParameter.Busy OR bExec_ParWritePers) THEN
		fbMcWriteParameter	( 	Axis 	:= AxisRef,
								Execute	:= bExec_ParWritePers );
	ELSE
		fbMcWriteParameter.Execute := FALSE ; 
		RETURN;
	END_IF
						
// fault handling 
	IF fbMcWriteParameter.Error THEN 
		bError					:= TRUE							;
		stFault.Active 			:= TRUE 						;
		stFault.MessageNumber	:= E_MessageNumbers.FF_AxisFault;
		stFault.Discription		:= CONCAT('Cannot write parameter Id#:', UDINT_TO_STRING(fbMcHome.ErrorID));
		stFault.Discription		:= CONCAT( sName , stfault.Discription ) ;
		stFault.FaultType		:= E_FaultTypes.FF				;
	END_IF
 
// reset commands
	bExec_ParWritePers := FALSE ;
END_METHOD

METHOD PUBLIC Init : BOOL
VAR_INPUT
	// Message location data
	nId			: UDINT ; // Identification number of object
	nParentId	: UDINT ; // Id of higher level If aplicable (0 = no parent)
	// Config Bits
	bIcfCmdVelocityRpm	: BOOL := FALSE ; // input speeds in Rpm
	bIcfEnableForward 	: BOOL := TRUE 	; // Enable forward motion
	bIcfEnablereverse	: BOOL := TRUE 	; // Enable reverse motion
	bIcfAlwaysEnable	: BOOL := FALSE ; // 1 = Axis always enabled, 0 = Axis disabled at Idle 
	bIcfSimulationMode	: BOOL := FALSE ; // Simulation mode is active [default set to False] Used for testing without hardware present 
	bIcfModuloAxis		: BOOL := FALSE ; // Show axis position as modulo
	bIcfSTOPresent		: BOOL := FALSE ; // Axis safe torque off is present
	bIcfNCHomeSensor	: BOOL := FALSE ; // Homing sensor is inverted (NC)	
	// Config Values 
	mcHomingMode 		: MC_HomingMode := MC_HomingMode.MC_DefaultHoming; 
	fHomePosition		: LREAL := 0 	; // set position at homing
	fSafeOverride		: LREAL := 10	; // Safe velocity override [%]
	nEncTurnoverVal 	: LREAL := 360	; // encoder turnover value 
	tEnableDelay		: time 	:= T#0MS; // Time between axis enable command and motion command execution (0 := no delay active)	
	tDisabledelay		: TIME 	:= T#100MS; // Axis idle time before axis is disabled 
END_VAR
VAR 
	bActVeloReadValid 	: BOOL ; // velocity parameter read is valid 
	bActAccReadValid 	: BOOL ; // Acceleration parameter read is valid 
	bActDecReadValid 	: BOOL ; // Deceleration parameter read is valid 
	bActParamValid 		: BOOL ; // Parameter read is valid 
END_VAR
// ====== Calculate device id =====
	ExecIdentifyDevice(nId,nParentId, E_ComponentTypes.Axis);

// ====== Set manual device type ======
	eDevType := E_Devices.Axis ;	
	
// ===== Message data set =====
	stFault.ComponentType		:= E_ComponentTypes.Axis ;
	
// ===== Read system configuration =====
	McReadSysVelo	(	Axis 			:= AxisRef,
						Enable 			:= Cmd_EnDriveParRead ,
						ParameterNumber := MaxVelocitySystem ,
						ReadMode		:= 1,
						Valid			=> bActVeloReadValid ,						
						Busy			=> ,
						Error			=> ,
						ErrorID			=> ,
						Value			=> fMaxVelo );
	McReadSysAcc	(	Axis 			:= AxisRef,
						Enable 			:= Cmd_EnDriveParRead ,
						ParameterNumber := MaxAccelerationSystem ,
						ReadMode		:= 1,
						Valid			=> bActAccReadValid ,						
						Busy			=> ,
						Error			=> ,
						ErrorID			=> ,
						Value			=> fMaxAcc );
	McReadSysDec	(	Axis 			:= AxisRef,
						Enable 			:= Cmd_EnDriveParRead ,
						ParameterNumber := MaxDecelerationSystem ,
						ReadMode		:= 1,
						Valid			=> bActDecReadValid ,						
						Busy			=> ,
						Error			=> ,
						ErrorID			=> ,
						Value			=> fMaxDec );

	IF 	fMaxVelo > 0 
	AND fMaxAcc >0
	AND fMaxDec >0 THEN 
		bActParamValid	:= TRUE ; 
		fCmdAcc 		:= fMaxAcc * 0.9;
		fCmdDecc		:= fMaxDec * 0.9;
	END_IF

	IF NOT Cmd_EnDriveParRead AND NOT bActParamValid THEN  
		Cmd_EnDriveParRead := TRUE;
	ELSIF Cmd_EnDriveParRead THEN
		Cmd_EnDriveParRead := FALSE;
	END_IF

// ===== Configure Axis =====
	// ***** Config Bits *****
		THIS^.bIcfCmdVelocityRpm	:= bIcfCmdVelocityRpm	; // Enable speed inputs in Rpm
		THIS^.bIcfEnableForward 	:= bIcfEnableForward 	; // Enable forward motion
		THIS^.bIcfEnablereverse		:= bIcfEnablereverse	; // Enable reverse motion
		THIS^.bIcfAlwaysEnable		:= bIcfAlwaysEnable		; // Always enable motor and brake if safety is ok
		THIS^.bIcfSimulationMode	:= bIcfSimulationMode 	; // Simulation mode is active [default set to False] 
		THIS^.bIcfModuloAxis		:= bIcfModuloAxis		; // show axis position as modulo
		THIS^.bIcfSTOPresent		:= bIcfSTOPresent		; // Axis has safe torque off function
		THIS^.bIcfNCHomeSensor		:= bIcfNCHomeSensor		; // Axis homing sensor is NC	
	// ***** config homing Mode ***** 
 		THIS^.mcHomingMode 			:= mcHomingMode ; // set homing mode
		THIS^.fHomePosition			:= fHomePosition;
	// ***** Velocity settings *****
		THIS^.fSafeOverride			:= fSafeOverride	; 	
	// ***** Encoder values *****
		THIS^.fEncoderTurnoverValue := nEncTurnoverVal	; // turnover value for encoder = 25.6 mm per rev * 4096 revolutions 
	// ***** Time delay enable off *****
		THIS^.tEnableDelay		:= tEnableDelay	;
		THIS^.tDisableDelay 	:= tDisabledelay ;		
		
// ===== configure parameters =====
	ParAccManualScaling.fMinimum 		:= 1 	;
	ParAccManualScaling.fMaximum		:= 100 	;
	ParAccManualScaling.nNumber 		:= nLocationId + 1;
	ParAccManualScaling.sDiscription  	:= CONCAT( STR1 := sName, STR2 := 'percantage of acceleration used For jogging');
	ParAccManualScaling.sName			:= CONCAT( STR1 := sName, STR2 := 'Manual acc scaling');
	ParAccManualScaling.sType			:= 'Mpar';
	ParAccManualScaling.sUnit			:= '%';

	ParDecManualScaling.fMinimum 		:= 1 	;
	ParDecManualScaling.fMaximum		:= 100 	;
	ParDecManualScaling.nNumber 		:= nLocationId + 2;
	ParDecManualScaling.sDiscription  	:= CONCAT( STR1 := sName, STR2 := 'percantage of deceleration used For jogging');
	ParDecManualScaling.sName			:= CONCAT( STR1 := sName, STR2 := 'Manual dec scaling');
	ParDecManualScaling.sType			:= 'Mpar';
	ParDecManualScaling.sUnit			:= '%';
		
// ===== reset axis state indicators ======
	bError 	:= FALSE;

// ====== Set init to done =======
IF bActParamValid THEN 
	bInitOk	:= TRUE ; 
END_IF
END_METHOD

END_FUNCTION_BLOCK

// ---- Buttons/Functions/FB_DevPushbuttonLight.TcPOU
{attribute 'reflection'}
FUNCTION_BLOCK PUBLIC FB_DevPushbuttonLight EXTENDS Fb_DevDigitalInputFunctions
VAR_OUTPUT
END_VAR
VAR
	fbLight : Fb_DevLight ; // light control 
END_VAR

// Set device type
IF eDevType = E_Devices.Undefined THEN 
	eDevType := E_Devices.PushButtonLight ;
END_IF

SUPER^(refFbFault := refFbFault);

// Light commands
	
fbLight(bEnable := bEnable, refFbFault := refFbFault);

METHOD PUBLIC CmdBlinkFast : BOOL
VAR_INPUT
END_VAR
CmdBlinkFast := fbLight.CmdBlinkFast();
END_METHOD

METHOD PUBLIC CmdBlinkSlow : BOOL
VAR_INPUT
END_VAR
CmdBlinkSlow	:= fbLight.CmdBlinkSlow();
END_METHOD

METHOD PUBLIC CmdOn : BOOL
VAR_INPUT
END_VAR
CmdOn := fbLight.CmdOn() ;
END_METHOD

END_FUNCTION_BLOCK

// ---- Lights/Functions/Fb_DevLight.TcPOU
{attribute 'reflection'}
FUNCTION_BLOCK PUBLIC Fb_DevLight EXTENDS FB_DevBase ;
VAR_OUTPUT
	bSoftLightOut	: BOOL ; // Software light output	
END_VAR
VAR
	bCmdBlinkSlow	: BOOL := FALSE ; // Command light blink slow
	bCmdBlinkFast 	: BOOL := FALSE ; // Command light blink fast
	bCmdOn			: BOOL := FALSE ; // Command turn light on	 
	qLight AT %Q* 	: BOOL := FALSE ; // light output
END_VAR

// set device type
IF eDevType = E_Devices.Undefined THEN 
	eDevType := E_Devices.DigitalOut ;
END_IF

// ===== check if light is enabled ======
	IF NOT bEnable AND NOT bCmdManual THEN 
		qLight := FALSE ;
		RETURN; 
	END_IF
	
// ===== set light output ======
	ExecSetOutput();

METHOD PUBLIC CmdBlinkFast : BOOL
VAR_INPUT
END_VAR
bCmdBlinkFast S= TRUE ;

CmdBlinkFast := bCmdBlinkFast ;
END_METHOD

METHOD PUBLIC CmdBlinkSlow : BOOL
VAR_INPUT
END_VAR
bCmdBlinkSlow S= TRUE ;

CmdBlinkSlow	:= bCmdBlinkSlow ;
END_METHOD

METHOD PUBLIC CmdOn : BOOL
VAR_INPUT
END_VAR
bCmdOn S= TRUE ;

CmdOn := qLight ;
END_METHOD

METHOD PRIVATE ExecSetOutput : BOOL
VAR_INPUT
END_VAR
// ===== set light output state =====
IF bCmdOn THEN 
	qLight S= TRUE ;
ELSIF bCmdBlinkFast THEN 
	qLight := Sys_Variables.BlinkFast 	;
ELSIF bCmdBlinkSlow THEN 
	qLight := Sys_Variables.BlinkSlow	;
ELSE
	qLight := FALSE ;
END_IF

// set soft output
bSoftLightOut	:= qLight;

// reset all commands 
bCmdOn			:= FALSE ;
bCmdBlinkFast 	:= FALSE ;
bCmdBlinkSlow 	:= FALSE ;
END_METHOD

METHOD PUBLIC Init : BOOL
VAR_INPUT
	// Location data for messages  
	nId			: UDINT ; // Identification number of object
	nParentId	: UDINT ; // Id of higher level If aplicable (0 = no parent)
END_VAR
// ====== Set init to true =====
	bInitOk	:= TRUE ; 

// ====== Calculate device id =====
	bInitOk :=	ExecIdentifyDevice(nId,nParentId, E_ComponentTypes.DiOutput) AND bInitOk;

// ===== Set feedback =====
	Init := bInitOk;
END_METHOD

END_FUNCTION_BLOCK

// ---- Sensors/AnalogInput/FunctionBlocks/FB_DevAnalogInput.TcPOU
{attribute 'reflection'}
FUNCTION_BLOCK PUBLIC FB_DevAnalogInput EXTENDS FB_DevBase
VAR_INPUT
	bCmdSimulate	: BOOL 	:= FALSE ;// Simulate sensor Input 
	fSimValue		: INT	:= 0 ;// Simulated sensor state
END_VAR
VAR_OUTPUT
	fValue	: LREAL := 0 ; // Input value from hardware (converted to LREAL)
END_VAR
VAR
	{attribute 'analysis' := '-33'}
	nLimitMin		: INT := Utilities_Library.GVL_FixedValues.nINTMINVALUE ; // Initial value is set to integer minimum value for use with normal def analog inputs 
	{attribute 'analysis' := '-33'}
	nLimitMax 		: INT := Utilities_Library.GVL_FixedValues.nINTMAXVALUE	; // Initial value is set to integer minimum value for use with high def analog inputs
	inHwInput AT%I* : INT ; // Hardware connection
END_VAR

// Set device type
eDevType := E_Devices.AnalogSensor ;

// Call base function
SUPER^(refFbFault := refFbFault);

// set feedback
ExecSetFeedback();

// Make sure compiler does not skip unused variables

METHOD ExecSetFeedback : BOOL
VAR_INPUT
END_VAR
IF bCmdSimulate THEN 
	fValue := int_to_lreal(fSimValue) ;
ELSE
	fValue := INT_TO_LREAL(inHwInput);
END_IF
END_METHOD

METHOD PUBLIC Init : BOOL
VAR_INPUT
	// Location data for messages  
	nId			: UDINT ; // Identification number of object
	nParentId	: UDINT ; // Id of higher level If aplicable (0 = no parent)
END_VAR
// ====== Calculate device id =====
	ExecIdentifyDevice(nId,nParentId, E_ComponentTypes.AnInput);

// ====== Set feedback ======
	bInitOk := true ;
END_METHOD

END_FUNCTION_BLOCK

// ---- Outputs/AnalogOutputs/FB_DevAnalogOutput.TcPOU
{attribute 'reflection'}
FUNCTION_BLOCK PUBLIC FB_DevAnalogOutput EXTENDS FB_DevBase 
VAR_INPUT
	fCmdValue		: LREAL := 0 ;
END_VAR
VAR_OUTPUT
	fOutputValue	: LREAL := 0 ;
END_VAR
VAR
	nLimitMin		: INT := -32767 ;
	nLimitMax 		: INT := 32767 ;
	qnHwOut	AT%Q*	: INT := 0 ;
END_VAR

// set device type
IF eDevType = E_Devices.Undefined THEN 
	eDevType := E_Devices.AnalogOut ;
END_IF

// Call base function
SUPER^(refFbFault := refFbFault);


// Call private functions
ExecSetOutput();
ExecSetFeedback();

METHOD INTERNAL ExecSetFeedback : BOOL
VAR_INPUT
END_VAR
// Set feedback 
fOutputValue := INT_TO_LREAL(qnHwOut) ;
END_METHOD

METHOD INTERNAL ExecSetOutput : BOOL
VAR_INPUT
END_VAR
// Set Output to physical device
IF bSafetyOk AND (bEnable OR bCmdManual) THEN 
	qnHwOut := LREAL_TO_INT(fCmdValue) ; 
	qnHwOut := LIMIT(nLimitMin, qnHwOut, nLimitMax) ; 
ELSE 
	qnHwOut 	:= 0;
	fCmdValue 	:= 0 ; 
END_IF
END_METHOD

METHOD PUBLIC Init : BOOL
VAR_INPUT
	// Location data for messages  
	nId				: UDINT; // Identification number of object
	nParentId		: UDINT; // Id of higher level If aplicable (0 = no parent)
	benableNegative	: BOOL ; // Enable negative values
END_VAR
// ====== Set init to true =====
	bInitOk	:= TRUE ; 

// ====== Calculate device id =====
	bInitOk :=	ExecIdentifyDevice(nId,nParentId, E_ComponentTypes.AnOutput) AND bInitOk;
	
// ====== set minimum value ========
	IF benableNegative THEN 
		nLimitMin := -32767;
	ELSE
		nLimitMin := 0 ;
	END_IF
	
// ====== Set feedback ======
	Init 	:= TRUE ;
END_METHOD

END_FUNCTION_BLOCK

// ---- Outputs/DigitalOutputs/FB_DevDigitalOutput.TcPOU
{attribute 'reflection'}
FUNCTION_BLOCK PUBLIC FB_DevDigitalOutput EXTENDS FB_DevBase
VAR_INPUT
	bCmdOn			: BOOL ; // command output status
END_VAR
VAR_OUTPUT
	bOutputState	: BOOL := FALSE ; // State of physical output
END_VAR
VAR
	qbOutput AT%Q* : BOOL ; // Output to physical device
END_VAR

// Call base function
SUPER^(refFbFault := refFbFault);


// Call private functions
ExecSetOutput();
ExecSetFeedback();

METHOD PRIVATE ExecSetFeedback : BOOL
VAR_INPUT
END_VAR
// Set feedback 
bOutputState := qbOutput ;
END_METHOD

METHOD PRIVATE ExecSetOutput : BOOL
VAR_INPUT
END_VAR
// Set Output to physical device
IF bSafetyOk AND (bEnable OR bCmdManual) THEN 
	qbOutput := bCmdOn ; 
ELSE 
	qbOutput S= FALSE ; 
END_IF
END_METHOD

METHOD PUBLIC Init : BOOL
VAR_INPUT
	// Location data for messages  
	nId			: UDINT ; // Identification number of object
	nParentId	: UDINT ; // Id of higher level If aplicable (0 = no parent)
END_VAR
// ====== Set init to true =====
	bInitOk	:= TRUE ; 

// ====== Calculate device id =====
	bInitOk :=	ExecIdentifyDevice(nId,nParentId, E_ComponentTypes.DiOutput) AND bInitOk;

// ====== Set feedback =====
	Init := bInitOk;
END_METHOD

END_FUNCTION_BLOCK

// ---- Heaters/FB_DevPWMGenerator.TcPOU
{attribute 'reflection'}
FUNCTION_BLOCK PUBLIC FB_DevPWMGenerator EXTENDS FB_DevBase
VAR_INPUT
	nPeriodLength	: DINT	:= 2000 ; // desired PWM cycle time length [ms] 
	nDutyCycle 		: DINT	:= 50 ; // percentage of power [%]
END_VAR
VAR_OUTPUT
END_VAR
VAR
	qbOutput	AT %Q* 	: BOOL 	; // physical output
	bCycleOutput		: BOOL 	; // Cycle output
	tonTimerOn  		: TON 	; // Timer for cycle on
	tofTimerOff			: TOF 	; // timer for cycle off 
	// output commands
	bCmdPWMCycle		: BOOL 	; // run PWM cycle 
	bCmdOn				: BOOL 	; // turn output on permanantly
END_VAR

// Set device type
eDevType := E_Devices.PWMController ;
SUPER^(refFbFault := refFbFault); 

// calculate cycle times 
CalcCycle();
// set outputs
ExecSetOutput(); 

// reset manual enable
bCmdManual := FALSE ;

METHOD PRIVATE CalcCycle : BOOL
VAR_INPUT
END_VAR
// check if dutycycle is within limits
nDutyCycle := LIMIT(1,nDutyCycle,100);

// Calculate time on from cycle time
tonTimerOn.PT 	:= DINT_TO_TIME(( nPeriodLength / 100) * nDutyCycle);
tofTimerOff.PT	:= DINT_TO_TIME(( nPeriodLength / 100) * (100 - nDutyCycle));
END_METHOD

METHOD PUBLIC CmdOutputCycle : BOOL // start PWM cycle stays on until off command is given
VAR_INPUT
END_VAR
bCmdPWMCycle 	S= TRUE ;
CmdOutputCycle 	:= bCmdPWMCycle ;
END_METHOD

METHOD PUBLIC CmdOutputOff : BOOL // turn off output signal completely
VAR_INPUT
END_VAR
bCmdPWMCycle 	:= FALSE ;
bCmdOn			:= FALSE ;
CmdOutputOff	:= TRUE 	;
END_METHOD

METHOD PUBLIC CmdOutputOn : BOOL // Output stays on until command ends (returns to PWM if active otherwise turns off)
VAR_INPUT
END_VAR
bCmdOn 		S= TRUE ;
CmdOutputOn	:= TRUE ;
END_METHOD

METHOD PRIVATE ExecSetOutput : BOOL
VAR_INPUT
END_VAR

// PWM signal generator
IF bCmdPWMCycle THEN 
	// Run cycle timers 
	tofTimerOff	(IN := tonTimerOn.Q);
	tonTimerOn	(IN := bCycleOutput AND NOT tofTimerOff.Q );
	bCycleOutput := NOT tofTimerOff.Q ;
ELSE
	bCycleOutput := FALSE ;
END_IF

// set output 
IF bSafetyOk AND (bEnable OR bCmdManual) THEN 
	qbOutput := bCycleOutput OR bCmdOn ;
ELSE
	qbOutput := FALSE ;
	RETURN; 
END_IF

// reset continuous on command
bCmdOn := false ;
END_METHOD

METHOD PUBLIC Init : BOOL
VAR_INPUT
	// Location data for messages  
	nId			: UDINT ; // Identification number of object
	nParentId	: UDINT ; // Id of higher level If aplicable (0 = no parent)
END_VAR
// ====== Set init to true =====
	bInitOk	:= TRUE ; 

// ====== Calculate device id =====
	bInitOk :=	ExecIdentifyDevice(nId,nParentId, E_ComponentTypes.Heaters) AND bInitOk;
END_METHOD

END_FUNCTION_BLOCK

// ---- Heaters/FB_DevDoublePWM.TcPOU
{attribute 'reflection'}
FUNCTION_BLOCK PUBLIC FB_DevDoublePWM EXTENDS FB_DevBase // PWM control for 2 outputs that cannot be switchid on simultaniously
VAR_INPUT
	bCmdPWMOn			: BOOL := FALSE ; // PWM controller on 
END_VAR
VAR_OUTPUT
END_VAR
VAR
	bCmdChanelAOn		: BOOL := FALSE ; // command switch chanel A on permanently
	bCmdChanelBOn		: BOOL := FALSE ; // Commandswitch chanel B on permanently 
	bCmdOverrulePWM		: BOOL := FALSE ; // Command to overrule PWM
	bCmdHold			: BOOL := false ; // Command hold PWM on signals (collision avoidance)

	tPeriodLength		: TIME  ; // desired PWM cycle time length [ms] 
	tDutyCycle 			: TIME	; // percentage of power [%]
	tIdleTime			: TIME	; // Time both outputs are idle during PWM
	
	tonOutputA 			: TON ; // Timer on PWM output A
	tonOutputB 			: TON ; // Timer on PWM output B
	tonIdle				: TON ; // Timer On PWM Idle time (both outputs off)

	tofOutputA 			: TOF ; // Timer off PWM output A Off (For overlap prevention)
	tofOutputB 			: TOF ; // Timer off PWM output B Off ( for overlap prevention)

	stParPeriodLength	: Udt_Parameter := (fValue := 2000); // desired PWM cycle time length [ms] Parameter
	stParDutyCycle 		: Udt_Parameter	:= ( fValue := 0); // percentage of power [%] Parameter
	stParSwitchOverTime	: Udt_Parameter	; // Time between switching A off and B on (and vice versa) Parameter
	stMaxTimeOn			: Udt_Parameter := (fValue := 1000);// Maximum time a heater can be on without burning through
	
	qbOutputMain AT %Q* 	: BOOL 	; // physical output to main relais
	qbOutputA	 AT %Q* 	: BOOL 	; // physical output to output A
	qbOutputB	 AT %Q* 	: BOOL 	; // physical output to output B
	
	nPWMStep	: INT ; // PWM stepper

	tonBurnTimeA	: TON ; // burn timer for coil A
	tonBurnTimeB	: TON ; // burn timer for coil B 
END_VAR

// set device type
IF eDevType = E_Devices.Undefined THEN 
	eDevType := E_Devices.DoublePWMController ;
END_IF

// Call base function
SUPER^(refFbFault := refFbFault);


// ===== hold all actions if not initialized ======
IF NOT bInitOk THEN
	RETURN;
END_IF 

// call Functions 
CalcCycleTimes();
IF tDutyCycle > T#0S AND tPeriodLength > T#0S THEN // switch PWM controller up when cycle timer is null
	ExecPWMCycle(); // 
END_IF 

ExecSetOutputs();

METHOD INTERNAL CalcCycleTimes : BOOL // calculate cycle timers
VAR_INPUT
END_VAR
VAR 
END_VAR
// Calculate Cycle timers
tPeriodLength	:= LREAL_TO_TIME( stParPeriodLength.fValue );
tDutyCycle		:= LREAL_TO_TIME(stParPeriodLength.fValue * (stParDutyCycle.fValue / 100));
tIdleTime		:= LREAL_TO_TIME(stParPeriodLength.fValue) - (tDutyCycle * 2) ;

tofOutputA.PT := LREAL_TO_TIME(stParSwitchOverTime.fValue);
tofOutputB.PT := LREAL_TO_TIME(stParSwitchOverTime.fValue);
END_METHOD

METHOD PUBLIC CmdHold : BOOL
VAR_INPUT
END_VAR
bCmdHold := TRUE ;

CmdHold := NOT qbOutputMain ;
END_METHOD

METHOD PUBLIC CmdOutputAOn : BOOL // Turn on chanel A permanently 
VAR_INPUT
END_VAR
bCmdOverrulePWM S= TRUE ;
bCmdChanelAOn S= TRUE ;

CmdOutputAOn := qbOutputA AND qbOutputMain ;
END_METHOD

METHOD PUBLIC CmdOutputBOn : BOOL
VAR_INPUT
END_VAR
bCmdOverrulePWM S= TRUE ;
bCmdChanelBOn S= TRUE ;

CmdOutputBOn := qbOutputB AND qbOutputMain ;
END_METHOD

METHOD PUBLIC CmdSafeStop : BOOL
VAR_INPUT
END_VAR
bCmdOverrulePWM S= TRUE ;
bCmdChanelAOn 		:= FALSE ;
bCmdChanelBOn		:= FALSE ;
qbOutputMain 		:= FALSE ;

bIsSafe := NOT (qbOutputA OR qbOutputB OR qbOutputMain);
END_METHOD

METHOD INTERNAL ExecPWMCycle : BOOL
VAR_INPUT
END_VAR
IF bCmdPWMOn THEN 
	IF bCmdOverrulePWM OR bCmdHold THEN 
		IF bCmdChanelAOn THEN 
			nPWMStep := 1 ;
		ELSE 
			nPWMStep := 0 ;
		END_IF
		bCmdOverrulePWM := FALSE ;
		RETURN;
	END_IF
ELSE 
	RETURN;
END_IF

// PWM stepper 
CASE nPWMStep OF 
	0: // Switch on chanel A
		bCmdChanelAOn := TRUE ;
		IF tonOutputA.Q THEN
			nPWMStep := 1 ;
		END_IF
	1: // Switch on chanel B
		bCmdChanelBOn := TRUE;
		IF tonOutputB.Q THEN
			nPWMStep := 2 ;
		END_IF
	2: // Idle Time 
		IF tonIdle.Q THEN 
			nPWMStep := 0;
		END_IF
	ELSE
		;
END_CASE

// call timers 
tonOutputA	(IN := bCmdChanelAOn, PT := tDutyCycle);
tonOutputB	(IN := bCmdChanelBOn, PT := tDutyCycle);
tonIdle 	(IN := nPWMStep = 2	, PT := tIdleTime);
END_METHOD

METHOD PRIVATE ExecSetOutputs : BOOL
VAR_INPUT
END_VAR

// Set main output
qbOutputMain := (bEnable OR bManual) AND bSafetyOk AND NOT bCmdHold ;

// Set outputs
qbOutputA := bCmdChanelAOn AND NOT tofOutputB.Q AND NOT tonBurnTimeA.Q;
qbOutputB := bCmdChanelBOn AND NOT tofOutputA.Q AND NOT tonBurnTimeB.Q;

// Call timers for overlap prevention
tofOutputA(IN := qbOutputA);
tofOutputB(IN := qbOutputB);

// reset commands
bCmdChanelAOn := FALSE ;
bCmdChanelBOn := FALSE ;

tonBurnTimeA ( IN := bCmdChanelAOn, PT := LREAL_TO_TIME( stMaxTimeOn.fValue));
tonBurnTimeB ( IN := bCmdChanelBOn, PT := LREAL_TO_TIME( stMaxTimeOn.fValue));

IF tonBurnTimeA.Q THEN 
	stFault.Active 			:= TRUE ;
	stFault.Discription 	:= 'Heater A burn timeout';
	stFault.MessageNumber 	:= E_MessageNumbers.CF_MoveToSlow ;
	stFault.FaultType		:= E_FaultTypes.CF;
	qbOutputA 				:= FALSE ;
ELSIF tonBurnTimeB.Q THEN 
	stFault.Active 			:= TRUE ;
	stFault.Discription 	:= 'Heater B burn timeout';
	stFault.MessageNumber 	:= E_MessageNumbers.CF_MoveToSlow ;
	stFault.FaultType		:= E_FaultTypes.CF;
	qbOutputB 				:= FALSE ;
END_IF

bCmdHold := FALSE ;
END_METHOD

METHOD PUBLIC Init : BOOL
VAR_INPUT
	// Message location data
	nId			: UDINT ; // Identification number of object
	nParentId	: UDINT ; // Id of higher level If aplicable (0 = no parent)
END_VAR
// ====== Calculate device id =====
	ExecIdentifyDevice(nId,nParentId, E_ComponentTypes.Heaters);

// ====== Set message information =======
	stFault.ComponentType	:= E_ComponentTypes.Heaters	;

// ======= Reset Error bit ======
	bErrorActive 	:= FALSE;
	bBussy			:= FALSE;
	
// ===== configure parameters =====
	stParPeriodLength.fMinimum 		:= 0 		;
	stParPeriodLength.fMaximum		:= 60000 	;
	stParPeriodLength.nNumber 		:= nLocationId + 1;
	stParPeriodLength.sDiscription  := CONCAT( STR1 := sName, STR2 := 'Period length of the cycle in miliseconds');
	stParPeriodLength.sName			:= CONCAT( STR1 := sName, STR2 := 'Period Length');
	stParPeriodLength.sType			:= 'MPar';
	stParPeriodLength.sUnit			:= 'ms';
	stParPeriodLength.fValue		:= 5000;

